LIN {X 0,Y 126.826,Z 270.322,A -85,B 0,C 180,E1 -25581.757,E2 -25581.757} C_VEL
LIN {X 0,Y 128.484,Z 273.393,A -85,B 0,C 180,E1 -25583.684,E2 -25583.684} C_VEL
LIN {X 0,Y 131.097,Z 275.877,A -85,B 0,C 180,E1 -25586.142,E2 -25586.142} C_VEL
LIN {X 0,Y 133.484,Z 279.395,A -85,B 0,C 180,E1 -25588.285,E2 -25588.285} C_VEL
LIN {X 0,Y 134.907,Z 280.969,A -85,B 0,C 180,E1 -25589.416,E2 -25589.416} C_VEL
LIN {X 0,Y 138.452,Z 286.009,A -85,B 0,C 180,E1 -25592.1,E2 -25592.1} C_VEL
LIN {X 0,Y 141.575,Z 290.551,A -85,B 0,C 180,E1 -25594.231,E2 -25594.231} C_VEL
LIN {X 0,Y 145.259,Z 296.604,A -85,B 0,C 180,E1 -25596.563,E2 -25596.563} C_VEL
LIN {X 0,Y 150.081,Z 307.019,A -85,B 0,C 180,E1 -25599.468,E2 -25599.468} C_VEL
LIN {X 0,Y 153.935,Z 317.286,A -85,B 0,C 180,E1 -25601.685,E2 -25601.685} C_VEL
LIN {X 0,Y 155.41,Z 322.258,A -85,B 0,C 180,E1 -25602.549,E2 -25602.549} C_VEL
LIN {X 0,Y 155.477,Z 325.681,A -85,B 0,C 180,E1 -25602.79,E2 -25602.79} C_VEL
LIN {X 0,Y 152.439,Z 367.811,A -85,B 0,C 180,E1 -25604.482,E2 -25604.482} C_VEL
LIN {X 0,Y 150.559,Z 380.968,A -85,B 0,C 180,E1 -25605.426,E2 -25605.426} C_VEL
LIN {X 0,Y 148.013,Z 393.091,A -85,B 0,C 180,E1 -25606.723,E2 -25606.723} C_VEL
LIN {X 0,Y 144.645,Z 405.228,A -85,B 0,C 180,E1 -25608.547,E2 -25608.547} C_VEL
LIN {X 0,Y 140.782,Z 416.789,A -85,B 0,C 180,E1 -25610.931,E2 -25610.931} C_VEL
LIN {X 0,Y 136.675,Z 427.192,A -85,B 0,C 180,E1 -25613.748,E2 -25613.748} C_VEL
LIN {X 0,Y 132.64,Z 436.533,A -85,B 0,C 180,E1 -25617.105,E2 -25617.105} C_VEL
LIN {X 0,Y 128.668,Z 445.603,A -85,B 0,C 180,E1 -25621.45,E2 -25621.45} C_VEL
LIN {X 0,Y 125.227,Z 452.89,A -85,B 0,C 180,E1 -25625.991,E2 -25625.991} C_VEL
LIN {X 0,Y 122.854,Z 457.8,A -85,B 0,C 180,E1 -25629.926,E2 -25629.926} C_VEL
LIN {X 0,Y 120.908,Z 462.575,A -85,B 0,C 180,E1 -25634.837,E2 -25634.837} C_VEL
LIN {X 0,Y 119.782,Z 466.223,A -85,B 0,C 180,E1 -25639.862,E2 -25639.862} C_VEL
LIN {X 0,Y 119.407,Z 468.103,A -85,B 0,C 180,E1 -25643.24,E2 -25643.24} C_VEL
LIN {X 0,Y 119.284,Z 469.509,A -85,B 0,C 180,E1 -25646.622,E2 -25646.622} C_VEL
LIN {X 0,Y 119.361,Z 470.506,A -85,B 0,C 180,E1 -25650,E2 -25650} C_VEL
LIN {X 0,Y 119.283,Z 471.098,A -85,B 0,C 180,E1 -25653.378,E2 -25653.378} C_VEL
LIN {X 0,Y 119.41,Z 471.3,A -85,B 0,C 180,E1 -25656.76,E2 -25656.76} C_VEL
LIN {X 0,Y 120.566,Z 470.457,A -85,B 0,C 180,E1 -25663.484,E2 -25663.484} C_VEL
LIN {X 0,Y 123.147,Z 468.068,A -85,B 0,C 180,E1 -25670.025,E2 -25670.025} C_VEL
LIN {X 0,Y 126.221,Z 465.155,A -85,B 0,C 180,E1 -25674.683,E2 -25674.683} C_VEL
LIN {X 0,Y 130.037,Z 461.227,A -85,B 0,C 180,E1 -25679.105,E2 -25679.105} C_VEL
LIN {X 0,Y 133.353,Z 457.578,A -85,B 0,C 180,E1 -25682.215,E2 -25682.215} C_VEL
LIN {X 0,Y 135.043,Z 454.869,A -85,B 0,C 180,E1 -25684.337,E2 -25684.337} C_VEL
LIN {X 0,Y 136.611,Z 450.087,A -85,B 0,C 180,E1 -25687.954,E2 -25687.954} C_VEL
LIN {X 0,Y 138.587,Z 444.753,A -85,B 0,C 180,E1 -25691.319,E2 -25691.319} C_VEL
LIN {X 0,Y 140.811,Z 441.114,A -85,B 0,C 180,E1 -25692.983,E2 -25692.983} C_VEL
LIN {X 0,Y 146.833,Z 432.313,A -85,B 0,C 180,E1 -25695.886,E2 -25695.886} C_VEL
LIN {X 0,Y 152.728,Z 422.206,A -85,B 0,C 180,E1 -25698.398,E2 -25698.398} C_VEL
LIN {X 0,Y 158.344,Z 410.772,A -85,B 0,C 180,E1 -25700.46,E2 -25700.46} C_VEL
LIN {X 0,Y 162.862,Z 399.545,A -85,B 0,C 180,E1 -25701.957,E2 -25701.957} C_VEL
LIN {X 0,Y 166.733,Z 386.906,A -85,B 0,C 180,E1 -25703.214,E2 -25703.214} C_VEL
LIN {X 0,Y 169.736,Z 373.483,A -85,B 0,C 180,E1 -25704.077,E2 -25704.077} C_VEL
LIN {X 0,Y 171.471,Z 360.998,A -85,B 0,C 180,E1 -25704.574,E2 -25704.574} C_VEL
LIN {X 0,Y 172.722,Z 344.57,A -85,B 0,C 180,E1 -25705.176,E2 -25705.176} C_VEL
LIN {X 0,Y 168.984,Z 334.445,A -85,B 0,C 180,E1 -25708.103,E2 -25708.103} C_VEL
LIN {X 0,Y 165.185,Z 325.649,A -85,B 0,C 180,E1 -25711.397,E2 -25711.397} C_VEL
LIN {X 0,Y 161.765,Z 318.418,A -85,B 0,C 180,E1 -25714.824,E2 -25714.824} C_VEL
LIN {X 0,Y 159.779,Z 315.16,A -85,B 0,C 180,E1 -25717.023,E2 -25717.023} C_VEL
LIN {X 0,Y 157.234,Z 311.251,A -85,B 0,C 180,E1 -25720.292,E2 -25720.292} C_VEL
LIN {X 0,Y 154.947,Z 307.802,A -85,B 0,C 180,E1 -25723.997,E2 -25723.997} C_VEL
LIN {X 0,Y 154.532,Z 306.974,A -85,B 0,C 180,E1 -25724.841,E2 -25724.841} C_VEL
LIN {X 0,Y 152.302,Z 304.116,A -85,B 0,C 180,E1 -25730.586,E2 -25730.586} C_VEL
LIN {X 0,Y 151.876,Z 301.949,A -85,B 0,C 180,E1 -25733.44,E2 -25733.44} C_VEL
LIN {X 0,Y 151.879,Z 301.933,A -85,B 0,C 180,E1 -25740.995,E2 -25740.995} C_VEL
LIN {X 0,Y 153.369,Z 305.636,A -85,B 0,C 180,E1 -25747.074,E2 -25747.074} C_VEL
LIN {X 0,Y 154.795,Z 307.238,A -85,B 0,C 180,E1 -25750.072,E2 -25750.072} C_VEL
LIN {X 0,Y 157.088,Z 310.973,A -85,B 0,C 180,E1 -25753.915,E2 -25753.915} C_VEL
LIN {X 0,Y 158.67,Z 313.546,A -85,B 0,C 180,E1 -25756.072,E2 -25756.072} C_VEL
LIN {X 0,Y 160.804,Z 316.708,A -85,B 0,C 180,E1 -25758.556,E2 -25758.556} C_VEL
LIN {X 0,Y 163.156,Z 320.534,A -85,B 0,C 180,E1 -25760.982,E2 -25760.982} C_VEL
LIN {X 0,Y 166.614,Z 326.408,A -85,B 0,C 180,E1 -25764.093,E2 -25764.093} C_VEL
LIN {X 0,Y 170.736,Z 334.213,A -85,B 0,C 180,E1 -25767.337,E2 -25767.337} C_VEL
LIN {X 0,Y 173.225,Z 339.607,A -85,B 0,C 180,E1 -25769.135,E2 -25769.135} C_VEL
LIN {X 0,Y 171.033,Z 362.908,A -85,B 0,C 180,E1 -25769.93,E2 -25769.93} C_VEL
LIN {X 0,Y 168.76,Z 375.767,A -85,B 0,C 180,E1 -25770.673,E2 -25770.673} C_VEL
LIN {X 0,Y 165.427,Z 388.725,A -85,B 0,C 180,E1 -25771.823,E2 -25771.823} C_VEL
LIN {X 0,Y 161.557,Z 399.746,A -85,B 0,C 180,E1 -25773.132,E2 -25773.132} C_VEL
LIN {X 0,Y 157.151,Z 409.955,A -85,B 0,C 180,E1 -25774.739,E2 -25774.739} C_VEL
LIN {X 0,Y 152.12,Z 419.837,A -85,B 0,C 180,E1 -25776.802,E2 -25776.802} C_VEL
LIN {X 0,Y 146.048,Z 430.047,A -85,B 0,C 180,E1 -25779.651,E2 -25779.651} C_VEL
LIN {X 0,Y 139.433,Z 439.163,A -85,B 0,C 180,E1 -25783.041,E2 -25783.041} C_VEL
LIN {X 0,Y 133.538,Z 446.491,A -85,B 0,C 180,E1 -25786.829,E2 -25786.829} C_VEL
LIN {X 0,Y 128.262,Z 452.341,A -85,B 0,C 180,E1 -25790.94,E2 -25790.94} C_VEL
LIN {X 0,Y 123.611,Z 456.926,A -85,B 0,C 180,E1 -25795.35,E2 -25795.35} C_VEL
LIN {X 0,Y 120.93,Z 459.336,A -85,B 0,C 180,E1 -25798.463,E2 -25798.463} C_VEL
LIN {X 0,Y 117.135,Z 462.465,A -85,B 0,C 180,E1 -25804.158,E2 -25804.158} C_VEL
LIN {X 0,Y 114.995,Z 463.953,A -85,B 0,C 180,E1 -25808.488,E2 -25808.488} C_VEL
LIN {X 0,Y 112.798,Z 464.935,A -85,B 0,C 180,E1 -25815.568,E2 -25815.568} C_VEL
LIN {X 0,Y 112.284,Z 464.849,A -85,B 0,C 180,E1 -25819.177,E2 -25819.177} C_VEL
LIN {X 0,Y 112.12,Z 464.344,A -85,B 0,C 180,E1 -25822.798,E2 -25822.798} C_VEL
LIN {X 0,Y 112.173,Z 463.43,A -85,B 0,C 180,E1 -25826.408,E2 -25826.408} C_VEL
LIN {X 0,Y 112.449,Z 462.131,A -85,B 0,C 180,E1 -25830,E2 -25830} C_VEL
LIN {X 0,Y 113.358,Z 459.394,A -85,B 0,C 180,E1 -25835.336,E2 -25835.336} C_VEL
LIN {X 0,Y 114.989,Z 455.651,A -85,B 0,C 180,E1 -25840.565,E2 -25840.565} C_VEL
LIN {X 0,Y 117.389,Z 450.796,A -85,B 0,C 180,E1 -25845.629,E2 -25845.629} C_VEL
LIN {X 0,Y 120.516,Z 444.687,A -85,B 0,C 180,E1 -25850.481,E2 -25850.481} C_VEL
LIN {X 0,Y 124.47,Z 437.084,A -85,B 0,C 180,E1 -25855.054,E2 -25855.054} C_VEL
LIN {X 0,Y 129.018,Z 427.533,A -85,B 0,C 180,E1 -25859.357,E2 -25859.357} C_VEL
LIN {X 0,Y 133.372,Z 417.674,A -85,B 0,C 180,E1 -25862.692,E2 -25862.692} C_VEL
LIN {X 0,Y 137.534,Z 406.586,A -85,B 0,C 180,E1 -25865.539,E2 -25865.539} C_VEL
LIN {X 0,Y 140.975,Z 395.728,A -85,B 0,C 180,E1 -25867.64,E2 -25867.64} C_VEL
LIN {X 0,Y 144.007,Z 383.744,A -85,B 0,C 180,E1 -25869.378,E2 -25869.378} C_VEL
LIN {X 0,Y 146.382,Z 371.309,A -85,B 0,C 180,E1 -25870.644,E2 -25870.644} C_VEL
LIN {X 0,Y 148,Z 357.95,A -85,B 0,C 180,E1 -25871.499,E2 -25871.499} C_VEL
LIN {X 0,Y 150.865,Z 319.683,A -85,B 0,C 180,E1 -25872.99,E2 -25872.99} C_VEL
LIN {X 0,Y 149.954,Z 317.15,A -85,B 0,C 180,E1 -25873.53,E2 -25873.53} C_VEL
LIN {X 0,Y 144.652,Z 306.547,A -85,B 0,C 180,E1 -25876.616,E2 -25876.616} C_VEL
LIN {X 0,Y 139.238,Z 297.373,A -85,B 0,C 180,E1 -25880.113,E2 -25880.113} C_VEL
LIN {X 0,Y 134.139,Z 289.816,A -85,B 0,C 180,E1 -25883.883,E2 -25883.883} C_VEL
LIN {X 0,Y 131.283,Z 285.807,A -85,B 0,C 180,E1 -25886.291,E2 -25886.291} C_VEL
LIN {X 0,Y 128.327,Z 281.654,A -85,B 0,C 180,E1 -25889.107,E2 -25889.107} C_VEL
LIN {X 0,Y 125.771,Z 278.792,A -85,B 0,C 180,E1 -25891.799,E2 -25891.799} C_VEL
LIN {X 0,Y 124.677,Z 276.71,A -85,B 0,C 180,E1 -25893.194,E2 -25893.194} C_VEL
LIN {X 0,Y 122.052,Z 274.673,A -85,B 0,C 180,E1 -25896.54,E2 -25896.54} C_VEL
LIN {X 0,Y 120.593,Z 271.942,A -85,B 0,C 180,E1 -25899.03,E2 -25899.03} C_VEL
LIN {X 0,Y 120.38,Z 271.211,A -85,B 0,C 180,E1 -25899.494,E2 -25899.494} C_VEL
LIN {X 0,Y 117.203,Z 269.28,A -85,B 0,C 180,E1 -25906.121,E2 -25906.121} C_VEL
LIN {X 0,Y 115.68,Z 266.37,A -85,B 0,C 180,E1 -25913.896,E2 -25913.896} C_VEL
LIN {X 0,Y 115.837,Z 265.042,A -85,B 0,C 180,E1 -25919.131,E2 -25919.131} C_VEL
LIN {X 0,Y 115.913,Z 265.227,A -85,B 0,C 180,E1 -25920.542,E2 -25920.542} C_VEL
LIN {X 0,Y 116.233,Z 267.39,A -85,B 0,C 180,E1 -25923.683,E2 -25923.683} C_VEL
LIN {X 0,Y 118.644,Z 270.26,A -85,B 0,C 180,E1 -25930.988,E2 -25930.988} C_VEL
LIN {X 0,Y 120.43,Z 271.31,A -85,B 0,C 180,E1 -25934.252,E2 -25934.252} C_VEL
LIN {X 0,Y 121.706,Z 274.109,A -85,B 0,C 180,E1 -25936.566,E2 -25936.566} C_VEL
LIN {X 0,Y 124.365,Z 276.547,A -85,B 0,C 180,E1 -25940.097,E2 -25940.097} C_VEL
LIN {X 0,Y 124.962,Z 277.268,A -85,B 0,C 180,E1 -25940.828,E2 -25940.828} C_VEL
LIN {X 0,Y 127.197,Z 280.647,A -85,B 0,C 180,E1 -25943.426,E2 -25943.426} C_VEL
LIN {X 0,Y 128.896,Z 282.384,A -85,B 0,C 180,E1 -25945.104,E2 -25945.104} C_VEL
LIN {X 0,Y 131.517,Z 286.037,A -85,B 0,C 180,E1 -25947.553,E2 -25947.553} C_VEL
LIN {X 0,Y 135.419,Z 291.569,A -85,B 0,C 180,E1 -25950.759,E2 -25950.759} C_VEL
LIN {X 0,Y 139.937,Z 298.477,A -85,B 0,C 180,E1 -25954.008,E2 -25954.008} C_VEL
LIN {X 0,Y 142.719,Z 303.955,A -85,B 0,C 180,E1 -25955.895,E2 -25955.895} C_VEL
LIN {X 0,Y 146.411,Z 312.55,A -85,B 0,C 180,E1 -25958.281,E2 -25958.281} C_VEL
LIN {X 0,Y 150.054,Z 323.022,A -85,B 0,C 180,E1 -25960.558,E2 -25960.558} C_VEL
LIN {X 0,Y 150.464,Z 324.735,A -85,B 0,C 180,E1 -25960.838,E2 -25960.838} C_VEL
LIN {X 0,Y 147.292,Z 367.734,A -85,B 0,C 180,E1 -25962.617,E2 -25962.617} C_VEL
LIN {X 0,Y 145.279,Z 381.195,A -85,B 0,C 180,E1 -25963.604,E2 -25963.604} C_VEL
LIN {X 0,Y 142.64,Z 393.137,A -85,B 0,C 180,E1 -25964.906,E2 -25964.906} C_VEL
LIN {X 0,Y 139.373,Z 404.404,A -85,B 0,C 180,E1 -25966.603,E2 -25966.603} C_VEL
LIN {X 0,Y 135.326,Z 416.082,A -85,B 0,C 180,E1 -25969.03,E2 -25969.03} C_VEL
LIN {X 0,Y 130.97,Z 426.57,A -85,B 0,C 180,E1 -25971.895,E2 -25971.895} C_VEL
LIN {X 0,Y 126.688,Z 436.011,A -85,B 0,C 180,E1 -25975.346,E2 -25975.346} C_VEL
LIN {X 0,Y 122.408,Z 445.135,A -85,B 0,C 180,E1 -25979.843,E2 -25979.843} C_VEL
LIN {X 0,Y 118.706,Z 452.469,A -85,B 0,C 180,E1 -25984.581,E2 -25984.581} C_VEL
LIN {X 0,Y 116.187,Z 457.424,A -85,B 0,C 180,E1 -25988.72,E2 -25988.72} C_VEL
LIN {X 0,Y 114.024,Z 462.236,A -85,B 0,C 180,E1 -25993.897,E2 -25993.897} C_VEL
LIN {X 0,Y 112.769,Z 465.921,A -85,B 0,C 180,E1 -25999.224,E2 -25999.224} C_VEL
LIN {X 0,Y 112.329,Z 467.821,A -85,B 0,C 180,E1 -26002.812,E2 -26002.812} C_VEL
LIN {X 0,Y 112.181,Z 469.257,A -85,B 0,C 180,E1 -26006.408,E2 -26006.408} C_VEL
LIN {X 0,Y 112.262,Z 470.27,A -85,B 0,C 180,E1 -26010,E2 -26010} C_VEL
LIN {X 0,Y 112.201,Z 470.878,A -85,B 0,C 180,E1 -26013.591,E2 -26013.591} C_VEL
LIN {X 0,Y 112.336,Z 471.098,A -85,B 0,C 180,E1 -26017.188,E2 -26017.188} C_VEL
LIN {X 0,Y 112.793,Z 470.9,A -85,B 0,C 180,E1 -26020.774,E2 -26020.774} C_VEL
LIN {X 0,Y 114.874,Z 469.316,A -85,B 0,C 180,E1 -26027.812,E2 -26027.812} C_VEL
LIN {X 0,Y 116.474,Z 467.943,A -85,B 0,C 180,E1 -26031.226,E2 -26031.226} C_VEL
LIN {X 0,Y 119.793,Z 465.063,A -85,B 0,C 180,E1 -26036.105,E2 -26036.105} C_VEL
LIN {X 0,Y 123.881,Z 461.17,A -85,B 0,C 180,E1 -26040.703,E2 -26040.703} C_VEL
LIN {X 0,Y 129.33,Z 455.389,A -85,B 0,C 180,E1 -26045.581,E2 -26045.581} C_VEL
LIN {X 0,Y 134.977,Z 448.685,A -85,B 0,C 180,E1 -26049.631,E2 -26049.631} C_VEL
LIN {X 0,Y 140.811,Z 441.114,A -85,B 0,C 180,E1 -26052.983,E2 -26052.983} C_VEL
LIN {X 0,Y 143.056,Z 437.279,A -85,B 0,C 180,E1 -26054.559,E2 -26054.559} C_VEL
LIN {X 0,Y 145.341,Z 430.766,A -85,B 0,C 180,E1 -26057.404,E2 -26057.404} C_VEL
LIN {X 0,Y 147.702,Z 423.796,A -85,B 0,C 180,E1 -26059.981,E2 -26059.981} C_VEL
LIN {X 0,Y 149.95,Z 419.15,A -85,B 0,C 180,E1 -26061.102,E2 -26061.102} C_VEL
LIN {X 0,Y 155.264,Z 408.282,A -85,B 0,C 180,E1 -26062.92,E2 -26062.92} C_VEL
LIN {X 0,Y 159.951,Z 396.309,A -85,B 0,C 180,E1 -26064.377,E2 -26064.377} C_VEL
LIN {X 0,Y 163.474,Z 384.532,A -85,B 0,C 180,E1 -26065.436,E2 -26065.436} C_VEL
LIN {X 0,Y 166.16,Z 372.192,A -85,B 0,C 180,E1 -26066.196,E2 -26066.196} C_VEL
LIN {X 0,Y 167.885,Z 359.393,A -85,B 0,C 180,E1 -26066.663,E2 -26066.663} C_VEL
LIN {X 0,Y 168.81,Z 347.255,A -85,B 0,C 180,E1 -26067.129,E2 -26067.129} C_VEL
LIN {X 0,Y 165.575,Z 338.228,A -85,B 0,C 180,E1 -26069.934,E2 -26069.934} C_VEL
LIN {X 0,Y 162.341,Z 330.413,A -85,B 0,C 180,E1 -26073.038,E2 -26073.038} C_VEL
LIN {X 0,Y 159.333,Z 323.765,A -85,B 0,C 180,E1 -26076.369,E2 -26076.369} C_VEL
LIN {X 0,Y 157.713,Z 321.142,A -85,B 0,C 180,E1 -26078.322,E2 -26078.322} C_VEL
LIN {X 0,Y 155.562,Z 317.639,A -85,B 0,C 180,E1 -26081.352,E2 -26081.352} C_VEL
LIN {X 0,Y 153.494,Z 314.14,A -85,B 0,C 180,E1 -26085.075,E2 -26085.075} C_VEL
LIN {X 0,Y 151.207,Z 310.7,A -85,B 0,C 180,E1 -26091.566,E2 -26091.566} C_VEL
LIN {X 0,Y 150.946,Z 308.985,A -85,B 0,C 180,E1 -26093.819,E2 -26093.819} C_VEL
LIN {X 0,Y 150.922,Z 308.838,A -85,B 0,C 180,E1 -26100.334,E2 -26100.334} C_VEL
LIN {X 0,Y 152.671,Z 313.002,A -85,B 0,C 180,E1 -26107.538,E2 -26107.538} C_VEL
LIN {X 0,Y 153.606,Z 314.216,A -85,B 0,C 180,E1 -26109.56,E2 -26109.56} C_VEL
LIN {X 0,Y 156.387,Z 318.86,A -85,B 0,C 180,E1 -26114.29,E2 -26114.29} C_VEL
LIN {X 0,Y 159.037,Z 323.21,A -85,B 0,C 180,E1 -26117.708,E2 -26117.708} C_VEL
LIN {X 0,Y 161.398,Z 327.222,A -85,B 0,C 180,E1 -26120.283,E2 -26120.283} C_VEL
LIN {X 0,Y 165.141,Z 334.046,A -85,B 0,C 180,E1 -26123.806,E2 -26123.806} C_VEL
LIN {X 0,Y 169.184,Z 342.339,A -85,B 0,C 180,E1 -26127.107,E2 -26127.107} C_VEL
LIN {X 0,Y 169.176,Z 344.32,A -85,B 0,C 180,E1 -26127.267,E2 -26127.267} C_VEL
LIN {X 0,Y 167.199,Z 363.569,A -85,B 0,C 180,E1 -26127.913,E2 -26127.913} C_VEL
LIN {X 0,Y 164.786,Z 376.603,A -85,B 0,C 180,E1 -26128.672,E2 -26128.672} C_VEL
LIN {X 0,Y 161.437,Z 389.043,A -85,B 0,C 180,E1 -26129.777,E2 -26129.777} C_VEL
LIN {X 0,Y 157.1,Z 400.836,A -85,B 0,C 180,E1 -26131.177,E2 -26131.177} C_VEL
LIN {X 0,Y 151.884,Z 412.18,A -85,B 0,C 180,E1 -26132.998,E2 -26132.998} C_VEL
LIN {X 0,Y 146.295,Z 422.366,A -85,B 0,C 180,E1 -26135.246,E2 -26135.246} C_VEL
LIN {X 0,Y 140.393,Z 431.524,A -85,B 0,C 180,E1 -26137.96,E2 -26137.96} C_VEL
LIN {X 0,Y 133.53,Z 440.421,A -85,B 0,C 180,E1 -26141.409,E2 -26141.409} C_VEL
LIN {X 0,Y 127.402,Z 447.526,A -85,B 0,C 180,E1 -26145.291,E2 -26145.291} C_VEL
LIN {X 0,Y 121.019,Z 453.995,A -85,B 0,C 180,E1 -26150.297,E2 -26150.297} C_VEL
LIN {X 0,Y 116.259,Z 458.238,A -85,B 0,C 180,E1 -26154.95,E2 -26154.95} C_VEL
LIN {X 0,Y 112.336,Z 461.4,A -85,B 0,C 180,E1 -26159.967,E2 -26159.967} C_VEL
LIN {X 0,Y 110.165,Z 462.965,A -85,B 0,C 180,E1 -26163.476,E2 -26163.476} C_VEL
LIN {X 0,Y 108.336,Z 464.107,A -85,B 0,C 180,E1 -26167.093,E2 -26167.093} C_VEL
LIN {X 0,Y 105.858,Z 465.125,A -85,B 0,C 180,E1 -26174.6,E2 -26174.6} C_VEL
LIN {X 0,Y 105.259,Z 465.056,A -85,B 0,C 180,E1 -26178.445,E2 -26178.445} C_VEL
LIN {X 0,Y 105.03,Z 464.586,A -85,B 0,C 180,E1 -26182.309,E2 -26182.309} C_VEL
LIN {X 0,Y 105.079,Z 463.689,A -85,B 0,C 180,E1 -26186.165,E2 -26186.165} C_VEL
LIN {X 0,Y 105.43,Z 462.132,A -85,B 0,C 180,E1 -26190.725,E2 -26190.725} C_VEL
LIN {X 0,Y 106.795,Z 458.606,A -85,B 0,C 180,E1 -26197.563,E2 -26197.563} C_VEL
LIN {X 0,Y 108.806,Z 454.547,A -85,B 0,C 180,E1 -26203.066,E2 -26203.066} C_VEL
LIN {X 0,Y 112.136,Z 448.329,A -85,B 0,C 180,E1 -26209.21,E2 -26209.21} C_VEL
LIN {X 0,Y 115.938,Z 441.559,A -85,B 0,C 180,E1 -26214.153,E2 -26214.153} C_VEL
LIN {X 0,Y 120.446,Z 433.123,A -85,B 0,C 180,E1 -26218.777,E2 -26218.777} C_VEL
LIN {X 0,Y 124.709,Z 424.451,A -85,B 0,C 180,E1 -26222.369,E2 -26222.369} C_VEL
LIN {X 0,Y 129.384,Z 413.777,A -85,B 0,C 180,E1 -26225.727,E2 -26225.727} C_VEL
LIN {X 0,Y 133.397,Z 403.133,A -85,B 0,C 180,E1 -26228.247,E2 -26228.247} C_VEL
LIN {X 0,Y 137.046,Z 391.213,A -85,B 0,C 180,E1 -26230.349,E2 -26230.349} C_VEL
LIN {X 0,Y 140.134,Z 378.16,A -85,B 0,C 180,E1 -26232.006,E2 -26232.006} C_VEL
LIN {X 0,Y 142.275,Z 365.227,A -85,B 0,C 180,E1 -26233.092,E2 -26233.092} C_VEL
LIN {X 0,Y 143.874,Z 347.807,A -85,B 0,C 180,E1 -26233.919,E2 -26233.919} C_VEL
LIN {X 0,Y 145.874,Z 321.687,A -85,B 0,C 180,E1 -26234.938,E2 -26234.938} C_VEL
LIN {X 0,Y 140.887,Z 311.337,A -85,B 0,C 180,E1 -26238.086,E2 -26238.086} C_VEL
LIN {X 0,Y 135.772,Z 302.426,A -85,B 0,C 180,E1 -26241.673,E2 -26241.673} C_VEL
LIN {X 0,Y 131.221,Z 295.406,A -85,B 0,C 180,E1 -26245.333,E2 -26245.333} C_VEL
LIN {X 0,Y 128.587,Z 291.604,A -85,B 0,C 180,E1 -26247.74,E2 -26247.74} C_VEL
LIN {X 0,Y 125.858,Z 287.692,A -85,B 0,C 180,E1 -26250.561,E2 -26250.561} C_VEL
LIN {X 0,Y 123.364,Z 284.409,A -85,B 0,C 180,E1 -26253.495,E2 -26253.495} C_VEL
LIN {X 0,Y 122.592,Z 283.199,A -85,B 0,C 180,E1 -26254.534,E2 -26254.534} C_VEL
LIN {X 0,Y 120.063,Z 280.701,A -85,B 0,C 180,E1 -26258.155,E2 -26258.155} C_VEL
LIN {X 0,Y 118.829,Z 278.036,A -85,B 0,C 180,E1 -26260.568,E2 -26260.568} C_VEL
LIN {X 0,Y 116.031,Z 276.032,A -85,B 0,C 180,E1 -26267.016,E2 -26267.016} C_VEL
LIN {X 0,Y 114.742,Z 272.986,A -85,B 0,C 180,E1 -26275.609,E2 -26275.609} C_VEL
LIN {X 0,Y 114.838,Z 272.283,A -85,B 0,C 180,E1 -26278.246,E2 -26278.246} C_VEL
LIN {X 0,Y 114.961,Z 272.627,A -85,B 0,C 180,E1 -26280.219,E2 -26280.219} C_VEL
LIN {X 0,Y 115.566,Z 275.123,A -85,B 0,C 180,E1 -26284.796,E2 -26284.796} C_VEL
LIN {X 0,Y 118.902,Z 278.148,A -85,B 0,C 180,E1 -26293.226,E2 -26293.226} C_VEL
LIN {X 0,Y 120.308,Z 280.999,A -85,B 0,C 180,E1 -26295.892,E2 -26295.892} C_VEL
LIN {X 0,Y 122.977,Z 283.651,A -85,B 0,C 180,E1 -26299.618,E2 -26299.618} C_VEL
LIN {X 0,Y 125.304,Z 287.177,A -85,B 0,C 180,E1 -26302.498,E2 -26302.498} C_VEL
LIN {X 0,Y 126.661,Z 288.694,A -85,B 0,C 180,E1 -26303.938,E2 -26303.938} C_VEL
LIN {X 0,Y 130.147,Z 293.716,A -85,B 0,C 180,E1 -26307.35,E2 -26307.35} C_VEL
LIN {X 0,Y 134.409,Z 300.046,A -85,B 0,C 180,E1 -26310.914,E2 -26310.914} C_VEL
LIN {X 0,Y 138.019,Z 306.426,A -85,B 0,C 180,E1 -26313.625,E2 -26313.625} C_VEL
LIN {X 0,Y 142.031,Z 315.996,A -85,B 0,C 180,E1 -26316.498,E2 -26316.498} C_VEL
LIN {X 0,Y 145.294,Z 325.657,A -85,B 0,C 180,E1 -26318.741,E2 -26318.741} C_VEL
LIN {X 0,Y 145.554,Z 327.024,A -85,B 0,C 180,E1 -26318.954,E2 -26318.954} C_VEL
LIN {X 0,Y 142.298,Z 367.725,A -85,B 0,C 180,E1 -26320.624,E2 -26320.624} C_VEL
LIN {X 0,Y 140.165,Z 381.308,A -85,B 0,C 180,E1 -26321.633,E2 -26321.633} C_VEL
LIN {X 0,Y 137.425,Z 393.168,A -85,B 0,C 180,E1 -26322.95,E2 -26322.95} C_VEL
LIN {X 0,Y 133.749,Z 405.168,A -85,B 0,C 180,E1 -26324.816,E2 -26324.816} C_VEL
LIN {X 0,Y 129.498,Z 416.667,A -85,B 0,C 180,E1 -26327.282,E2 -26327.282} C_VEL
LIN {X 0,Y 124.945,Z 427.017,A -85,B 0,C 180,E1 -26330.221,E2 -26330.221} C_VEL
LIN {X 0,Y 120.043,Z 437.132,A -85,B 0,C 180,E1 -26334.165,E2 -26334.165} C_VEL
LIN {X 0,Y 116.234,Z 444.69,A -85,B 0,C 180,E1 -26338.077,E2 -26338.077} C_VEL
LIN {X 0,Y 112.88,Z 450.921,A -85,B 0,C 180,E1 -26342.163,E2 -26342.163} C_VEL
LIN {X 0,Y 109.581,Z 457.048,A -85,B 0,C 180,E1 -26347.368,E2 -26347.368} C_VEL
LIN {X 0,Y 107.182,Z 461.898,A -85,B 0,C 180,E1 -26352.839,E2 -26352.839} C_VEL
LIN {X 0,Y 105.788,Z 465.619,A -85,B 0,C 180,E1 -26358.504,E2 -26358.504} C_VEL
LIN {X 0,Y 105.272,Z 467.536,A -85,B 0,C 180,E1 -26362.327,E2 -26362.327} C_VEL
LIN {X 0,Y 105.097,Z 469.005,A -85,B 0,C 180,E1 -26366.166,E2 -26366.166} C_VEL
LIN {X 0,Y 105.175,Z 470.034,A -85,B 0,C 180,E1 -26370,E2 -26370} C_VEL
LIN {X 0,Y 105.11,Z 470.657,A -85,B 0,C 180,E1 -26373.834,E2 -26373.834} C_VEL
LIN {X 0,Y 105.279,Z 470.893,A -85,B 0,C 180,E1 -26377.673,E2 -26377.673} C_VEL
LIN {X 0,Y 105.813,Z 470.727,A -85,B 0,C 180,E1 -26381.494,E2 -26381.494} C_VEL
LIN {X 0,Y 108.094,Z 469.174,A -85,B 0,C 180,E1 -26388.971,E2 -26388.971} C_VEL
LIN {X 0,Y 109.864,Z 467.818,A -85,B 0,C 180,E1 -26392.571,E2 -26392.571} C_VEL
LIN {X 0,Y 113.445,Z 464.972,A -85,B 0,C 180,E1 -26397.686,E2 -26397.686} C_VEL
LIN {X 0,Y 117.83,Z 461.116,A -85,B 0,C 180,E1 -26402.467,E2 -26402.467} C_VEL
LIN {X 0,Y 123.398,Z 455.619,A -85,B 0,C 180,E1 -26407.324,E2 -26407.324} C_VEL
LIN {X 0,Y 129.579,Z 448.734,A -85,B 0,C 180,E1 -26411.637,E2 -26411.637} C_VEL
LIN {X 0,Y 136.123,Z 440.679,A -85,B 0,C 180,E1 -26415.228,E2 -26415.228} C_VEL
LIN {X 0,Y 141.992,Z 432.472,A -85,B 0,C 180,E1 -26417.939,E2 -26417.939} C_VEL
LIN {X 0,Y 148.123,Z 422.467,A -85,B 0,C 180,E1 -26420.445,E2 -26420.445} C_VEL
LIN {X 0,Y 149.95,Z 419.15,A -85,B 0,C 180,E1 -26421.102,E2 -26421.102} C_VEL
LIN {X 0,Y 151.272,Z 415.992,A -85,B 0,C 180,E1 -26421.879,E2 -26421.879} C_VEL
LIN {X 0,Y 152.049,Z 411.02,A -85,B 0,C 180,E1 -26423.59,E2 -26423.59} C_VEL
LIN {X 0,Y 152.725,Z 405.872,A -85,B 0,C 180,E1 -26425.227,E2 -26425.227} C_VEL
LIN {X 0,Y 153.819,Z 402.439,A -85,B 0,C 180,E1 -26425.866,E2 -26425.866} C_VEL
LIN {X 0,Y 158.343,Z 389.577,A -85,B 0,C 180,E1 -26427.197,E2 -26427.197} C_VEL
LIN {X 0,Y 161.594,Z 377.163,A -85,B 0,C 180,E1 -26428.077,E2 -26428.077} C_VEL
LIN {X 0,Y 163.819,Z 364.366,A -85,B 0,C 180,E1 -26428.632,E2 -26428.632} C_VEL
LIN {X 0,Y 165.152,Z 350.219,A -85,B 0,C 180,E1 -26429.116,E2 -26429.116} C_VEL
LIN {X 0,Y 162.501,Z 342.549,A -85,B 0,C 180,E1 -26431.67,E2 -26431.67} C_VEL
LIN {X 0,Y 159.515,Z 334.863,A -85,B 0,C 180,E1 -26434.876,E2 -26434.876} C_VEL
LIN {X 0,Y 157.119,Z 329.345,A -85,B 0,C 180,E1 -26437.827,E2 -26437.827} C_VEL
LIN {X 0,Y 154.158,Z 324.328,A -85,B 0,C 180,E1 -26442.086,E2 -26442.086} C_VEL
LIN {X 0,Y 152.056,Z 320.673,A -85,B 0,C 180,E1 -26446.203,E2 -26446.203} C_VEL
LIN {X 0,Y 150.198,Z 317.48,A -85,B 0,C 180,E1 -26452.269,E2 -26452.269} C_VEL
LIN {X 0,Y 150.017,Z 316.064,A -85,B 0,C 180,E1 -26454.203,E2 -26454.203} C_VEL
LIN {X 0,Y 150.037,Z 316.031,A -85,B 0,C 180,E1 -26460.336,E2 -26460.336} C_VEL
LIN {X 0,Y 151.622,Z 319.95,A -85,B 0,C 180,E1 -26467.156,E2 -26467.156} C_VEL
LIN {X 0,Y 152.358,Z 320.985,A -85,B 0,C 180,E1 -26468.862,E2 -26468.862} C_VEL
LIN {X 0,Y 154.81,Z 325.331,A -85,B 0,C 180,E1 -26473.371,E2 -26473.371} C_VEL
LIN {X 0,Y 157.484,Z 329.95,A -85,B 0,C 180,E1 -26477.051,E2 -26477.051} C_VEL
LIN {X 0,Y 160.28,Z 335.032,A -85,B 0,C 180,E1 -26480.222,E2 -26480.222} C_VEL
LIN {X 0,Y 163.88,Z 342.223,A -85,B 0,C 180,E1 -26483.712,E2 -26483.712} C_VEL
LIN {X 0,Y 165.532,Z 345.865,A -85,B 0,C 180,E1 -26485.163,E2 -26485.163} C_VEL
LIN {X 0,Y 163.511,Z 364.721,A -85,B 0,C 180,E1 -26485.827,E2 -26485.827} C_VEL
LIN {X 0,Y 160.945,Z 377.768,A -85,B 0,C 180,E1 -26486.598,E2 -26486.598} C_VEL
LIN {X 0,Y 157.302,Z 390.362,A -85,B 0,C 180,E1 -26487.725,E2 -26487.725} C_VEL
LIN {X 0,Y 152.846,Z 401.928,A -85,B 0,C 180,E1 -26489.116,E2 -26489.116} C_VEL
LIN {X 0,Y 147.445,Z 413.097,A -85,B 0,C 180,E1 -26490.91,E2 -26490.91} C_VEL
LIN {X 0,Y 142.139,Z 422.353,A -85,B 0,C 180,E1 -26492.949,E2 -26492.949} C_VEL
LIN {X 0,Y 136.108,Z 431.361,A -85,B 0,C 180,E1 -26495.584,E2 -26495.584} C_VEL
LIN {X 0,Y 130.065,Z 438.958,A -85,B 0,C 180,E1 -26498.418,E2 -26498.418} C_VEL
LIN {X 0,Y 123.431,Z 446.392,A -85,B 0,C 180,E1 -26502.251,E2 -26502.251} C_VEL
LIN {X 0,Y 117.41,Z 452.337,A -85,B 0,C 180,E1 -26506.499,E2 -26506.499} C_VEL
LIN {X 0,Y 112.051,Z 457.011,A -85,B 0,C 180,E1 -26511.155,E2 -26511.155} C_VEL
LIN {X 0,Y 107.479,Z 460.56,A -85,B 0,C 180,E1 -26516.233,E2 -26516.233} C_VEL
LIN {X 0,Y 103.786,Z 463.083,A -85,B 0,C 180,E1 -26521.705,E2 -26521.705} C_VEL
LIN {X 0,Y 101.752,Z 464.255,A -85,B 0,C 180,E1 -26525.517,E2 -26525.517} C_VEL
LIN {X 0,Y 98.952,Z 465.315,A -85,B 0,C 180,E1 -26533.495,E2 -26533.495} C_VEL
LIN {X 0,Y 98.264,Z 465.263,A -85,B 0,C 180,E1 -26537.61,E2 -26537.61} C_VEL
LIN {X 0,Y 97.94,Z 464.822,A -85,B 0,C 180,E1 -26541.748,E2 -26541.748} C_VEL
LIN {X 0,Y 97.958,Z 463.949,A -85,B 0,C 180,E1 -26545.886,E2 -26545.886} C_VEL
LIN {X 0,Y 98.431,Z 462.114,A -85,B 0,C 180,E1 -26551.584,E2 -26551.584} C_VEL
LIN {X 0,Y 99.77,Z 458.938,A -85,B 0,C 180,E1 -26558.099,E2 -26558.099} C_VEL
LIN {X 0,Y 101.929,Z 454.919,A -85,B 0,C 180,E1 -26563.965,E2 -26563.965} C_VEL
LIN {X 0,Y 105.486,Z 448.746,A -85,B 0,C 180,E1 -26570.474,E2 -26570.474} C_VEL
LIN {X 0,Y 109.509,Z 442.025,A -85,B 0,C 180,E1 -26575.67,E2 -26575.67} C_VEL
LIN {X 0,Y 114.311,Z 433.673,A -85,B 0,C 180,E1 -26580.48,E2 -26580.48} C_VEL
LIN {X 0,Y 118.807,Z 425.073,A -85,B 0,C 180,E1 -26584.192,E2 -26584.192} C_VEL
LIN {X 0,Y 123.713,Z 414.487,A -85,B 0,C 180,E1 -26587.64,E2 -26587.64} C_VEL
LIN {X 0,Y 127.915,Z 403.968,A -85,B 0,C 180,E1 -26590.209,E2 -26590.209} C_VEL
LIN {X 0,Y 131.748,Z 392.277,A -85,B 0,C 180,E1 -26592.335,E2 -26592.335} C_VEL
LIN {X 0,Y 134.991,Z 379.433,A -85,B 0,C 180,E1 -26594.015,E2 -26594.015} C_VEL
LIN {X 0,Y 137.364,Z 366.121,A -85,B 0,C 180,E1 -26595.189,E2 -26595.189} C_VEL
LIN {X 0,Y 138.972,Z 350.08,A -85,B 0,C 180,E1 -26595.975,E2 -26595.975} C_VEL
LIN {X 0,Y 141.052,Z 324.264,A -85,B 0,C 180,E1 -26596.98,E2 -26596.98} C_VEL
LIN {X 0,Y 136.315,Z 314.404,A -85,B 0,C 180,E1 -26600.293,E2 -26600.293} C_VEL
LIN {X 0,Y 131.443,Z 305.718,A -85,B 0,C 180,E1 -26604.133,E2 -26604.133} C_VEL
LIN {X 0,Y 126.82,Z 298.42,A -85,B 0,C 180,E1 -26608.407,E2 -26608.407} C_VEL
LIN {X 0,Y 123.714,Z 293.998,A -85,B 0,C 180,E1 -26611.794,E2 -26611.794} C_VEL
LIN {X 0,Y 120.737,Z 289.719,A -85,B 0,C 180,E1 -26615.71,E2 -26615.71} C_VEL
LIN {X 0,Y 118.312,Z 286.978,A -85,B 0,C 180,E1 -26619.551,E2 -26619.551} C_VEL
LIN {X 0,Y 117.292,Z 284.835,A -85,B 0,C 180,E1 -26621.727,E2 -26621.727} C_VEL
LIN {X 0,Y 114.912,Z 282.866,A -85,B 0,C 180,E1 -26627.819,E2 -26627.819} C_VEL
LIN {X 0,Y 113.871,Z 279.882,A -85,B 0,C 180,E1 -26636.461,E2 -26636.461} C_VEL
LIN {X 0,Y 114.049,Z 280.09,A -85,B 0,C 180,E1 -26640.275,E2 -26640.275} C_VEL
LIN {X 0,Y 115.275,Z 283.135,A -85,B 0,C 180,E1 -26647.003,E2 -26647.003} C_VEL
LIN {X 0,Y 117.467,Z 284.985,A -85,B 0,C 180,E1 -26652.269,E2 -26652.269} C_VEL
LIN {X 0,Y 119.143,Z 288.136,A -85,B 0,C 180,E1 -26655.558,E2 -26655.558} C_VEL
LIN {X 0,Y 121.22,Z 290.346,A -85,B 0,C 180,E1 -26658.622,E2 -26658.622} C_VEL
LIN {X 0,Y 123.747,Z 294.017,A -85,B 0,C 180,E1 -26661.888,E2 -26661.888} C_VEL
LIN {X 0,Y 124.991,Z 295.832,A -85,B 0,C 180,E1 -26663.315,E2 -26663.315} C_VEL
LIN {X 0,Y 127.818,Z 299.964,A -85,B 0,C 180,E1 -26666.233,E2 -26666.233} C_VEL
LIN {X 0,Y 131.725,Z 306.128,A -85,B 0,C 180,E1 -26669.745,E2 -26669.745} C_VEL
LIN {X 0,Y 134.87,Z 312.023,A -85,B 0,C 180,E1 -26672.298,E2 -26672.298} C_VEL
LIN {X 0,Y 138.38,Z 321.061,A -85,B 0,C 180,E1 -26675.05,E2 -26675.05} C_VEL
LIN {X 0,Y 140.714,Z 328.397,A -85,B 0,C 180,E1 -26676.823,E2 -26676.823} C_VEL
LIN {X 0,Y 137.577,Z 367.067,A -85,B 0,C 180,E1 -26678.451,E2 -26678.451} C_VEL
LIN {X 0,Y 135.363,Z 380.646,A -85,B 0,C 180,E1 -26679.439,E2 -26679.439} C_VEL
LIN {X 0,Y 132.375,Z 393.188,A -85,B 0,C 180,E1 -26680.839,E2 -26680.839} C_VEL
LIN {X 0,Y 128.812,Z 404.334,A -85,B 0,C 180,E1 -26682.561,E2 -26682.561} C_VEL
LIN {X 0,Y 124.345,Z 415.95,A -85,B 0,C 180,E1 -26685.049,E2 -26685.049} C_VEL
LIN {X 0,Y 119.567,Z 426.396,A -85,B 0,C 180,E1 -26688.04,E2 -26688.04} C_VEL
LIN {X 0,Y 115.227,Z 434.938,A -85,B 0,C 180,E1 -26691.305,E2 -26691.305} C_VEL
LIN {X 0,Y 110.36,Z 443.871,A -85,B 0,C 180,E1 -26695.88,E2 -26695.88} C_VEL
LIN {X 0,Y 107.374,Z 449.359,A -85,B 0,C 180,E1 -26699.518,E2 -26699.518} C_VEL
LIN {X 0,Y 104.16,Z 454.775,A -85,B 0,C 180,E1 -26703.987,E2 -26703.987} C_VEL
LIN {X 0,Y 101.096,Z 460.074,A -85,B 0,C 180,E1 -26709.66,E2 -26709.66} C_VEL
LIN {X 0,Y 99.213,Z 464.198,A -85,B 0,C 180,E1 -26715.645,E2 -26715.645} C_VEL
LIN {X 0,Y 98.218,Z 467.25,A -85,B 0,C 180,E1 -26721.772,E2 -26721.772} C_VEL
LIN {X 0,Y 98.012,Z 468.752,A -85,B 0,C 180,E1 -26725.888,E2 -26725.888} C_VEL
LIN {X 0,Y 98.079,Z 469.798,A -85,B 0,C 180,E1 -26730,E2 -26730} C_VEL
LIN {X 0,Y 98.021,Z 470.437,A -85,B 0,C 180,E1 -26734.112,E2 -26734.112} C_VEL
LIN {X 0,Y 98.247,Z 470.689,A -85,B 0,C 180,E1 -26738.226,E2 -26738.226} C_VEL
LIN {X 0,Y 98.834,Z 470.549,A -85,B 0,C 180,E1 -26742.318,E2 -26742.318} C_VEL
LIN {X 0,Y 101.367,Z 469.033,A -85,B 0,C 180,E1 -26750.283,E2 -26750.283} C_VEL
LIN {X 0,Y 103.329,Z 467.694,A -85,B 0,C 180,E1 -26754.085,E2 -26754.085} C_VEL
LIN {X 0,Y 107.195,Z 464.882,A -85,B 0,C 180,E1 -26759.454,E2 -26759.454} C_VEL
LIN {X 0,Y 111.902,Z 461.061,A -85,B 0,C 180,E1 -26764.42,E2 -26764.42} C_VEL
LIN {X 0,Y 117.249,Z 456.134,A -85,B 0,C 180,E1 -26769.002,E2 -26769.002} C_VEL
LIN {X 0,Y 123.279,Z 449.949,A -85,B 0,C 180,E1 -26773.165,E2 -26773.165} C_VEL
LIN {X 0,Y 130.019,Z 442.264,A -85,B 0,C 180,E1 -26776.863,E2 -26776.863} C_VEL
LIN {X 0,Y 137.336,Z 432.632,A -85,B 0,C 180,E1 -26780.14,E2 -26780.14} C_VEL
LIN {X 0,Y 143.72,Z 422.707,A -85,B 0,C 180,E1 -26782.621,E2 -26782.621} C_VEL
LIN {X 0,Y 149.738,Z 411.515,A -85,B 0,C 180,E1 -26784.637,E2 -26784.637} C_VEL
LIN {X 0,Y 153.819,Z 402.439,A -85,B 0,C 180,E1 -26785.866,E2 -26785.866} C_VEL
LIN {X 0,Y 155.562,Z 397.209,A -85,B 0,C 180,E1 -26786.649,E2 -26786.649} C_VEL
LIN {X 0,Y 157.023,Z 388.583,A -85,B 0,C 180,E1 -26788.36,E2 -26788.36} C_VEL
LIN {X 0,Y 157.992,Z 379.693,A -85,B 0,C 180,E1 -26789.921,E2 -26789.921} C_VEL
LIN {X 0,Y 158.888,Z 374.047,A -85,B 0,C 180,E1 -26790.459,E2 -26790.459} C_VEL
LIN {X 0,Y 160.954,Z 360.844,A -85,B 0,C 180,E1 -26790.962,E2 -26790.962} C_VEL
LIN {X 0,Y 161.642,Z 353.043,A -85,B 0,C 180,E1 -26791.251,E2 -26791.251} C_VEL
LIN {X 0,Y 159.037,Z 345.172,A -85,B 0,C 180,E1 -26794.11,E2 -26794.11} C_VEL
LIN {X 0,Y 156.174,Z 337.638,A -85,B 0,C 180,E1 -26797.685,E2 -26797.685} C_VEL
LIN {X 0,Y 154.94,Z 334.831,A -85,B 0,C 180,E1 -26799.421,E2 -26799.421} C_VEL
LIN {X 0,Y 152.714,Z 330.951,A -85,B 0,C 180,E1 -26802.94,E2 -26802.94} C_VEL
LIN {X 0,Y 150.875,Z 327.496,A -85,B 0,C 180,E1 -26806.857,E2 -26806.857} C_VEL
LIN {X 0,Y 149.223,Z 324.292,A -85,B 0,C 180,E1 -26812.899,E2 -26812.899} C_VEL
LIN {X 0,Y 149.101,Z 323.097,A -85,B 0,C 180,E1 -26814.591,E2 -26814.591} C_VEL
LIN {X 0,Y 149.122,Z 323.087,A -85,B 0,C 180,E1 -26820,E2 -26820} C_VEL
LIN {X 0,Y 150.587,Z 326.893,A -85,B 0,C 180,E1 -26826.785,E2 -26826.785} C_VEL
LIN {X 0,Y 151.222,Z 327.958,A -85,B 0,C 180,E1 -26828.372,E2 -26828.372} C_VEL
LIN {X 0,Y 153.377,Z 332.037,A -85,B 0,C 180,E1 -26832.614,E2 -26832.614} C_VEL
LIN {X 0,Y 155.523,Z 335.934,A -85,B 0,C 180,E1 -26835.816,E2 -26835.816} C_VEL
LIN {X 0,Y 158.205,Z 341.102,A -85,B 0,C 180,E1 -26839.125,E2 -26839.125} C_VEL
LIN {X 0,Y 161.827,Z 348.848,A -85,B 0,C 180,E1 -26842.892,E2 -26842.892} C_VEL
LIN {X 0,Y 162.014,Z 349.294,A -85,B 0,C 180,E1 -26843.073,E2 -26843.073} C_VEL
LIN {X 0,Y 160.067,Z 365.737,A -85,B 0,C 180,E1 -26843.636,E2 -26843.636} C_VEL
LIN {X 0,Y 157.618,Z 377.692,A -85,B 0,C 180,E1 -26844.336,E2 -26844.336} C_VEL
LIN {X 0,Y 154.113,Z 389.69,A -85,B 0,C 180,E1 -26845.377,E2 -26845.377} C_VEL
LIN {X 0,Y 149.489,Z 401.43,A -85,B 0,C 180,E1 -26846.714,E2 -26846.714} C_VEL
LIN {X 0,Y 143.895,Z 412.735,A -85,B 0,C 180,E1 -26848.461,E2 -26848.461} C_VEL
LIN {X 0,Y 137.782,Z 422.98,A -85,B 0,C 180,E1 -26850.67,E2 -26850.67} C_VEL
LIN {X 0,Y 130.775,Z 432.835,A -85,B 0,C 180,E1 -26853.593,E2 -26853.593} C_VEL
LIN {X 0,Y 124.506,Z 440.216,A -85,B 0,C 180,E1 -26856.451,E2 -26856.451} C_VEL
LIN {X 0,Y 117.588,Z 447.462,A -85,B 0,C 180,E1 -26860.355,E2 -26860.355} C_VEL
LIN {X 0,Y 112.246,Z 452.38,A -85,B 0,C 180,E1 -26864.007,E2 -26864.007} C_VEL
LIN {X 0,Y 106.539,Z 457.051,A -85,B 0,C 180,E1 -26868.726,E2 -26868.726} C_VEL
LIN {X 0,Y 101.576,Z 460.64,A -85,B 0,C 180,E1 -26873.977,E2 -26873.977} C_VEL
LIN {X 0,Y 97.248,Z 463.36,A -85,B 0,C 180,E1 -26880.14,E2 -26880.14} C_VEL
LIN {X 0,Y 93.452,Z 465.153,A -85,B 0,C 180,E1 -26887.912,E2 -26887.912} C_VEL
LIN {X 0,Y 91.261,Z 465.47,A -85,B 0,C 180,E1 -26896.642,E2 -26896.642} C_VEL
LIN {X 0,Y 90.879,Z 465.052,A -85,B 0,C 180,E1 -26901.102,E2 -26901.102} C_VEL
LIN {X 0,Y 90.864,Z 464.207,A -85,B 0,C 180,E1 -26905.564,E2 -26905.564} C_VEL
LIN {X 0,Y 91.467,Z 462.011,A -85,B 0,C 180,E1 -26912.7,E2 -26912.7} C_VEL
LIN {X 0,Y 93.403,Z 458.035,A -85,B 0,C 180,E1 -26920.842,E2 -26920.842} C_VEL
LIN {X 0,Y 96.018,Z 453.688,A -85,B 0,C 180,E1 -26927.024,E2 -26927.024} C_VEL
LIN {X 0,Y 99.538,Z 448.159,A -85,B 0,C 180,E1 -26932.851,E2 -26932.851} C_VEL
LIN {X 0,Y 103.983,Z 441.259,A -85,B 0,C 180,E1 -26938.237,E2 -26938.237} C_VEL
LIN {X 0,Y 109.017,Z 432.885,A -85,B 0,C 180,E1 -26943.041,E2 -26943.041} C_VEL
LIN {X 0,Y 114.043,Z 423.754,A -85,B 0,C 180,E1 -26946.931,E2 -26946.931} C_VEL
LIN {X 0,Y 118.739,Z 414.028,A -85,B 0,C 180,E1 -26950.066,E2 -26950.066} C_VEL
LIN {X 0,Y 123.181,Z 403.342,A -85,B 0,C 180,E1 -26952.65,E2 -26952.65} C_VEL
LIN {X 0,Y 127.226,Z 391.362,A -85,B 0,C 180,E1 -26954.774,E2 -26954.774} C_VEL
LIN {X 0,Y 130.296,Z 379.526,A -85,B 0,C 180,E1 -26956.313,E2 -26956.313} C_VEL
LIN {X 0,Y 132.647,Z 367.009,A -85,B 0,C 180,E1 -26957.431,E2 -26957.431} C_VEL
LIN {X 0,Y 134.274,Z 352.266,A -85,B 0,C 180,E1 -26958.179,E2 -26958.179} C_VEL
LIN {X 0,Y 136.339,Z 326.795,A -85,B 0,C 180,E1 -26959.214,E2 -26959.214} C_VEL
LIN {X 0,Y 132.419,Z 318.457,A -85,B 0,C 180,E1 -26962.262,E2 -26962.262} C_VEL
LIN {X 0,Y 128.272,Z 310.84,A -85,B 0,C 180,E1 -26965.869,E2 -26965.869} C_VEL
LIN {X 0,Y 124.188,Z 304.134,A -85,B 0,C 180,E1 -26970.019,E2 -26970.019} C_VEL
LIN {X 0,Y 121.624,Z 300.232,A -85,B 0,C 180,E1 -26973.086,E2 -26973.086} C_VEL
LIN {X 0,Y 119.033,Z 296.327,A -85,B 0,C 180,E1 -26976.777,E2 -26976.777} C_VEL
LIN {X 0,Y 116.672,Z 293.321,A -85,B 0,C 180,E1 -26980.906,E2 -26980.906} C_VEL
LIN {X 0,Y 115.845,Z 291.596,A -85,B 0,C 180,E1 -26982.845,E2 -26982.845} C_VEL
LIN {X 0,Y 113.668,Z 289.412,A -85,B 0,C 180,E1 -26989.31,E2 -26989.31} C_VEL
LIN {X 0,Y 112.996,Z 287.003,A -85,B 0,C 180,E1 -26996.434,E2 -26996.434} C_VEL
LIN {X 0,Y 113.129,Z 287.11,A -85,B 0,C 180,E1 -26999.777,E2 -26999.777} C_VEL
LIN {X 0,Y 114.267,Z 290.128,A -85,B 0,C 180,E1 -27006.622,E2 -27006.622} C_VEL
LIN {X 0,Y 116.033,Z 291.719,A -85,B 0,C 180,E1 -27011.203,E2 -27011.203} C_VEL
LIN {X 0,Y 117.959,Z 295.174,A -85,B 0,C 180,E1 -27015.164,E2 -27015.164} C_VEL
LIN {X 0,Y 119.472,Z 296.916,A -85,B 0,C 180,E1 -27017.539,E2 -27017.539} C_VEL
LIN {X 0,Y 122.629,Z 301.707,A -85,B 0,C 180,E1 -27021.813,E2 -27021.813} C_VEL
LIN {X 0,Y 125.689,Z 306.491,A -85,B 0,C 180,E1 -27025.236,E2 -27025.236} C_VEL
LIN {X 0,Y 129.412,Z 312.797,A -85,B 0,C 180,E1 -27028.814,E2 -27028.814} C_VEL
LIN {X 0,Y 131.485,Z 316.977,A -85,B 0,C 180,E1 -27030.645,E2 -27030.645} C_VEL
LIN {X 0,Y 134.681,Z 325.718,A -85,B 0,C 180,E1 -27033.407,E2 -27033.407} C_VEL
LIN {X 0,Y 136.103,Z 330.438,A -85,B 0,C 180,E1 -27034.611,E2 -27034.611} C_VEL
LIN {X 0,Y 133.003,Z 366.965,A -85,B 0,C 180,E1 -27036.167,E2 -27036.167} C_VEL
LIN {X 0,Y 130.817,Z 379.999,A -85,B 0,C 180,E1 -27037.112,E2 -27037.112} C_VEL
LIN {X 0,Y 127.799,Z 392.093,A -85,B 0,C 180,E1 -27038.405,E2 -27038.405} C_VEL
LIN {X 0,Y 124.114,Z 403.499,A -85,B 0,C 180,E1 -27040.143,E2 -27040.143} C_VEL
LIN {X 0,Y 119.415,Z 415.235,A -85,B 0,C 180,E1 -27042.636,E2 -27042.636} C_VEL
LIN {X 0,Y 114.388,Z 425.773,A -85,B 0,C 180,E1 -27045.663,E2 -27045.663} C_VEL
LIN {X 0,Y 109.739,Z 434.382,A -85,B 0,C 180,E1 -27048.971,E2 -27048.971} C_VEL
LIN {X 0,Y 105.171,Z 442.327,A -85,B 0,C 180,E1 -27053.028,E2 -27053.028} C_VEL
LIN {X 0,Y 100.514,Z 450.081,A -85,B 0,C 180,E1 -27058.372,E2 -27058.372} C_VEL
LIN {X 0,Y 96.557,Z 456.289,A -85,B 0,C 180,E1 -27064.106,E2 -27064.106} C_VEL
LIN {X 0,Y 93.609,Z 461.216,A -85,B 0,C 180,E1 -27070.254,E2 -27070.254} C_VEL
LIN {X 0,Y 91.843,Z 465.011,A -85,B 0,C 180,E1 -27076.729,E2 -27076.729} C_VEL
LIN {X 0,Y 91.169,Z 466.963,A -85,B 0,C 180,E1 -27081.131,E2 -27081.131} C_VEL
LIN {X 0,Y 90.921,Z 468.493,A -85,B 0,C 180,E1 -27085.567,E2 -27085.567} C_VEL
LIN {X 0,Y 90.978,Z 469.561,A -85,B 0,C 180,E1 -27090,E2 -27090} C_VEL
LIN {X 0,Y 90.929,Z 470.216,A -85,B 0,C 180,E1 -27094.433,E2 -27094.433} C_VEL
LIN {X 0,Y 91.213,Z 470.484,A -85,B 0,C 180,E1 -27098.865,E2 -27098.865} C_VEL
LIN {X 0,Y 91.886,Z 470.366,A -85,B 0,C 180,E1 -27103.265,E2 -27103.265} C_VEL
LIN {X 0,Y 94.703,Z 468.891,A -85,B 0,C 180,E1 -27111.781,E2 -27111.781} C_VEL
LIN {X 0,Y 99.57,Z 465.849,A -85,B 0,C 180,E1 -27119.61,E2 -27119.61} C_VEL
LIN {X 0,Y 104.303,Z 462.405,A -85,B 0,C 180,E1 -27124.941,E2 -27124.941} C_VEL
LIN {X 0,Y 110.008,Z 457.732,A -85,B 0,C 180,E1 -27129.948,E2 -27129.948} C_VEL
LIN {X 0,Y 117.073,Z 451.092,A -85,B 0,C 180,E1 -27134.859,E2 -27134.859} C_VEL
LIN {X 0,Y 124.057,Z 443.716,A -85,B 0,C 180,E1 -27138.645,E2 -27138.645} C_VEL
LIN {X 0,Y 131.614,Z 434.569,A -85,B 0,C 180,E1 -27141.965,E2 -27141.965} C_VEL
LIN {X 0,Y 138.859,Z 424.007,A -85,B 0,C 180,E1 -27144.699,E2 -27144.699} C_VEL
LIN {X 0,Y 145.083,Z 413.265,A -85,B 0,C 180,E1 -27146.679,E2 -27146.679} C_VEL
LIN {X 0,Y 150.019,Z 402.824,A -85,B 0,C 180,E1 -27148.117,E2 -27148.117} C_VEL
LIN {X 0,Y 154.628,Z 390.291,A -85,B 0,C 180,E1 -27149.398,E2 -27149.398} C_VEL
LIN {X 0,Y 158.24,Z 377.069,A -85,B 0,C 180,E1 -27150.321,E2 -27150.321} C_VEL
LIN {X 0,Y 158.888,Z 374.047,A -85,B 0,C 180,E1 -27150.459,E2 -27150.459} C_VEL
LIN {X 0,Y 159.626,Z 368.687,A -85,B 0,C 180,E1 -27150.873,E2 -27150.873} C_VEL
LIN {X 0,Y 159.7,Z 363.502,A -85,B 0,C 180,E1 -27151.561,E2 -27151.561} C_VEL
LIN {X 0,Y 159.151,Z 358.804,A -85,B 0,C 180,E1 -27152.535,E2 -27152.535} C_VEL
LIN {X 0,Y 158.042,Z 354.938,A -85,B 0,C 180,E1 -27153.848,E2 -27153.848} C_VEL
LIN {X 0,Y 155.591,Z 347.397,A -85,B 0,C 180,E1 -27156.983,E2 -27156.983} C_VEL
LIN {X 0,Y 153.496,Z 341.635,A -85,B 0,C 180,E1 -27160.091,E2 -27160.091} C_VEL
LIN {X 0,Y 151.223,Z 337.373,A -85,B 0,C 180,E1 -27163.982,E2 -27163.982} C_VEL
LIN {X 0,Y 149.738,Z 334.342,A -85,B 0,C 180,E1 -27167.463,E2 -27167.463} C_VEL
LIN {X 0,Y 148.249,Z 331.021,A -85,B 0,C 180,E1 -27173.706,E2 -27173.706} C_VEL
LIN {X 0,Y 148.199,Z 330.233,A -85,B 0,C 180,E1 -27174.795,E2 -27174.795} C_VEL
LIN {X 0,Y 148.195,Z 330.09,A -85,B 0,C 180,E1 -27179.433,E2 -27179.433} C_VEL
LIN {X 0,Y 149.978,Z 334.618,A -85,B 0,C 180,E1 -27187.552,E2 -27187.552} C_VEL
LIN {X 0,Y 151.996,Z 338.763,A -85,B 0,C 180,E1 -27191.883,E2 -27191.883} C_VEL
LIN {X 0,Y 154.044,Z 342.725,A -85,B 0,C 180,E1 -27195.145,E2 -27195.145} C_VEL
LIN {X 0,Y 156.579,Z 348.082,A -85,B 0,C 180,E1 -27198.482,E2 -27198.482} C_VEL
LIN {X 0,Y 158.652,Z 352.755,A -85,B 0,C 180,E1 -27200.841,E2 -27200.841} C_VEL
LIN {X 0,Y 156.809,Z 367.135,A -85,B 0,C 180,E1 -27201.374,E2 -27201.374} C_VEL
LIN {X 0,Y 153.91,Z 380.036,A -85,B 0,C 180,E1 -27202.171,E2 -27202.171} C_VEL
LIN {X 0,Y 150.052,Z 392.018,A -85,B 0,C 180,E1 -27203.194,E2 -27203.194} C_VEL
LIN {X 0,Y 144.975,Z 404.11,A -85,B 0,C 180,E1 -27204.639,E2 -27204.639} C_VEL
LIN {X 0,Y 139.202,Z 414.84,A -85,B 0,C 180,E1 -27206.342,E2 -27206.342} C_VEL
LIN {X 0,Y 132.469,Z 425.289,A -85,B 0,C 180,E1 -27208.662,E2 -27208.662} C_VEL
LIN {X 0,Y 125.606,Z 434.311,A -85,B 0,C 180,E1 -27211.43,E2 -27211.43} C_VEL
LIN {X 0,Y 117.857,Z 442.731,A -85,B 0,C 180,E1 -27214.921,E2 -27214.921} C_VEL
LIN {X 0,Y 110.745,Z 449.487,A -85,B 0,C 180,E1 -27218.977,E2 -27218.977} C_VEL
LIN {X 0,Y 103.242,Z 455.662,A -85,B 0,C 180,E1 -27224.375,E2 -27224.375} C_VEL
LIN {X 0,Y 97.539,Z 459.654,A -85,B 0,C 180,E1 -27229.573,E2 -27229.573} C_VEL
LIN {X 0,Y 94.252,Z 461.699,A -85,B 0,C 180,E1 -27233.378,E2 -27233.378} C_VEL
LIN {X 0,Y 90.705,Z 463.679,A -85,B 0,C 180,E1 -27238.464,E2 -27238.464} C_VEL
LIN {X 0,Y 86.851,Z 465.325,A -85,B 0,C 180,E1 -27246.134,E2 -27246.134} C_VEL
LIN {X 0,Y 84.298,Z 465.678,A -85,B 0,C 180,E1 -27255.516,E2 -27255.516} C_VEL
LIN {X 0,Y 83.818,Z 465.277,A -85,B 0,C 180,E1 -27260.346,E2 -27260.346} C_VEL
LIN {X 0,Y 83.762,Z 464.466,A -85,B 0,C 180,E1 -27265.187,E2 -27265.187} C_VEL
LIN {X 0,Y 84.513,Z 462.015,A -85,B 0,C 180,E1 -27273.696,E2 -27273.696} C_VEL
LIN {X 0,Y 86.446,Z 458.367,A -85,B 0,C 180,E1 -27281.727,E2 -27281.727} C_VEL
LIN {X 0,Y 89.264,Z 454.061,A -85,B 0,C 180,E1 -27288.356,E2 -27288.356} C_VEL
LIN {X 0,Y 93.046,Z 448.577,A -85,B 0,C 180,E1 -27294.546,E2 -27294.546} C_VEL
LIN {X 0,Y 97.796,Z 441.731,A -85,B 0,C 180,E1 -27300.202,E2 -27300.202} C_VEL
LIN {X 0,Y 102.894,Z 433.894,A -85,B 0,C 180,E1 -27304.95,E2 -27304.95} C_VEL
LIN {X 0,Y 108.468,Z 424.377,A -85,B 0,C 180,E1 -27309.178,E2 -27309.178} C_VEL
LIN {X 0,Y 113.993,Z 413.567,A -85,B 0,C 180,E1 -27312.701,E2 -27312.701} C_VEL
LIN {X 0,Y 118.674,Z 402.659,A -85,B 0,C 180,E1 -27315.288,E2 -27315.288} C_VEL
LIN {X 0,Y 122.934,Z 390.446,A -85,B 0,C 180,E1 -27317.396,E2 -27317.396} C_VEL
LIN {X 0,Y 126.143,Z 378.415,A -85,B 0,C 180,E1 -27318.892,E2 -27318.892} C_VEL
LIN {X 0,Y 128.513,Z 365.627,A -85,B 0,C 180,E1 -27319.962,E2 -27319.962} C_VEL
LIN {X 0,Y 130.318,Z 348.512,A -85,B 0,C 180,E1 -27320.764,E2 -27320.764} C_VEL
LIN {X 0,Y 131.909,Z 329.53,A -85,B 0,C 180,E1 -27321.546,E2 -27321.546} C_VEL
LIN {X 0,Y 128.356,Z 321.857,A -85,B 0,C 180,E1 -27324.648,E2 -27324.648} C_VEL
LIN {X 0,Y 124.109,Z 313.858,A -85,B 0,C 180,E1 -27328.886,E2 -27328.886} C_VEL
LIN {X 0,Y 120.838,Z 308.48,A -85,B 0,C 180,E1 -27332.74,E2 -27332.74} C_VEL
LIN {X 0,Y 119.41,Z 306.222,A -85,B 0,C 180,E1 -27334.678,E2 -27334.678} C_VEL
LIN {X 0,Y 117.257,Z 302.782,A -85,B 0,C 180,E1 -27338.068,E2 -27338.068} C_VEL
LIN {X 0,Y 115.016,Z 299.459,A -85,B 0,C 180,E1 -27342.512,E2 -27342.512} C_VEL
LIN {X 0,Y 114.461,Z 298.408,A -85,B 0,C 180,E1 -27343.935,E2 -27343.935} C_VEL
LIN {X 0,Y 112.115,Z 294.172,A -85,B 0,C 180,E1 -27356.406,E2 -27356.406} C_VEL
LIN {X 0,Y 112.219,Z 294.162,A -85,B 0,C 180,E1 -27359.327,E2 -27359.327} C_VEL
LIN {X 0,Y 113.242,Z 297.077,A -85,B 0,C 180,E1 -27366.145,E2 -27366.145} C_VEL
LIN {X 0,Y 114.74,Z 298.62,A -85,B 0,C 180,E1 -27370.365,E2 -27370.365} C_VEL
LIN {X 0,Y 116.78,Z 302.209,A -85,B 0,C 180,E1 -27374.763,E2 -27374.763} C_VEL
LIN {X 0,Y 117.791,Z 303.52,A -85,B 0,C 180,E1 -27376.464,E2 -27376.464} C_VEL
LIN {X 0,Y 120.52,Z 307.885,A -85,B 0,C 180,E1 -27380.48,E2 -27380.48} C_VEL
LIN {X 0,Y 124.045,Z 313.637,A -85,B 0,C 180,E1 -27384.677,E2 -27384.677} C_VEL
LIN {X 0,Y 127.838,Z 320.93,A -85,B 0,C 180,E1 -27388.528,E2 -27388.528} C_VEL
LIN {X 0,Y 130.755,Z 329.329,A -85,B 0,C 180,E1 -27391.357,E2 -27391.357} C_VEL
LIN {X 0,Y 131.699,Z 332.556,A -85,B 0,C 180,E1 -27392.252,E2 -27392.252} C_VEL
LIN {X 0,Y 128.589,Z 367.248,A -85,B 0,C 180,E1 -27393.741,E2 -27393.741} C_VEL
LIN {X 0,Y 126.115,Z 380.861,A -85,B 0,C 180,E1 -27394.718,E2 -27394.718} C_VEL
LIN {X 0,Y 122.868,Z 393.209,A -85,B 0,C 180,E1 -27396.104,E2 -27396.104} C_VEL
LIN {X 0,Y 118.368,Z 405.85,A -85,B 0,C 180,E1 -27398.122,E2 -27398.122} C_VEL
LIN {X 0,Y 113.493,Z 417.118,A -85,B 0,C 180,E1 -27400.662,E2 -27400.662} C_VEL
LIN {X 0,Y 108.83,Z 426.222,A -85,B 0,C 180,E1 -27403.407,E2 -27403.407} C_VEL
LIN {X 0,Y 103.431,Z 435.557,A -85,B 0,C 180,E1 -27407.197,E2 -27407.197} C_VEL
LIN {X 0,Y 98.02,Z 444.209,A -85,B 0,C 180,E1 -27412.064,E2 -27412.064} C_VEL
LIN {X 0,Y 94.535,Z 449.661,A -85,B 0,C 180,E1 -27416.112,E2 -27416.112} C_VEL
LIN {X 0,Y 90.199,Z 455.911,A -85,B 0,C 180,E1 -27422.128,E2 -27422.128} C_VEL
LIN {X 0,Y 86.924,Z 460.875,A -85,B 0,C 180,E1 -27428.664,E2 -27428.664} C_VEL
LIN {X 0,Y 84.927,Z 464.707,A -85,B 0,C 180,E1 -27435.626,E2 -27435.626} C_VEL
LIN {X 0,Y 84.148,Z 466.677,A -85,B 0,C 180,E1 -27440.384,E2 -27440.384} C_VEL
LIN {X 0,Y 83.825,Z 468.228,A -85,B 0,C 180,E1 -27445.191,E2 -27445.191} C_VEL
LIN {X 0,Y 83.884,Z 469.325,A -85,B 0,C 180,E1 -27450,E2 -27450} C_VEL
LIN {X 0,Y 83.862,Z 469.996,A -85,B 0,C 180,E1 -27454.807,E2 -27454.807} C_VEL
LIN {X 0,Y 84.185,Z 470.278,A -85,B 0,C 180,E1 -27459.612,E2 -27459.612} C_VEL
LIN {X 0,Y 84.976,Z 470.179,A -85,B 0,C 180,E1 -27464.366,E2 -27464.366} C_VEL
LIN {X 0,Y 86.3,Z 469.67,A -85,B 0,C 180,E1 -27469.011,E2 -27469.011} C_VEL
LIN {X 0,Y 90.535,Z 467.445,A -85,B 0,C 180,E1 -27477.76,E2 -27477.76} C_VEL
LIN {X 0,Y 95.024,Z 464.701,A -85,B 0,C 180,E1 -27483.69,E2 -27483.69} C_VEL
LIN {X 0,Y 100.471,Z 460.953,A -85,B 0,C 180,E1 -27489.018,E2 -27489.018} C_VEL
LIN {X 0,Y 106.566,Z 456.101,A -85,B 0,C 180,E1 -27493.826,E2 -27493.826} C_VEL
LIN {X 0,Y 113.324,Z 450.004,A -85,B 0,C 180,E1 -27498.091,E2 -27498.091} C_VEL
LIN {X 0,Y 120.772,Z 442.439,A -85,B 0,C 180,E1 -27501.776,E2 -27501.776} C_VEL
LIN {X 0,Y 127.369,Z 434.718,A -85,B 0,C 180,E1 -27504.477,E2 -27504.477} C_VEL
LIN {X 0,Y 134.88,Z 424.244,A -85,B 0,C 180,E1 -27507.162,E2 -27507.162} C_VEL
LIN {X 0,Y 141.318,Z 413.591,A -85,B 0,C 180,E1 -27509.079,E2 -27509.079} C_VEL
LIN {X 0,Y 146.408,Z 403.296,A -85,B 0,C 180,E1 -27510.465,E2 -27510.465} C_VEL
LIN {X 0,Y 151.158,Z 391.007,A -85,B 0,C 180,E1 -27511.702,E2 -27511.702} C_VEL
LIN {X 0,Y 154.906,Z 377.927,A -85,B 0,C 180,E1 -27512.604,E2 -27512.604} C_VEL
LIN {X 0,Y 157.41,Z 365.076,A -85,B 0,C 180,E1 -27513.135,E2 -27513.135} C_VEL
LIN {X 0,Y 158.355,Z 355.959,A -85,B 0,C 180,E1 -27513.476,E2 -27513.476} C_VEL
LIN {X 0,Y 158.042,Z 354.938,A -85,B 0,C 180,E1 -27513.848,E2 -27513.848} C_VEL
LIN {X 0,Y 156.44,Z 351.873,A -85,B 0,C 180,E1 -27515.61,E2 -27515.61} C_VEL
LIN {X 0,Y 154.742,Z 349.633,A -85,B 0,C 180,E1 -27517.55,E2 -27517.55} C_VEL
LIN {X 0,Y 149.972,Z 344.168,A -85,B 0,C 180,E1 -27524.634,E2 -27524.634} C_VEL
LIN {X 0,Y 148.504,Z 341.048,A -85,B 0,C 180,E1 -27528.397,E2 -27528.397} C_VEL
LIN {X 0,Y 147.306,Z 337.747,A -85,B 0,C 180,E1 -27534.525,E2 -27534.525} C_VEL
LIN {X 0,Y 147.257,Z 337.127,A -85,B 0,C 180,E1 -27535.894,E2 -27535.894} C_VEL
LIN {X 0,Y 147.32,Z 337.318,A -85,B 0,C 180,E1 -27539.572,E2 -27539.572} C_VEL
LIN {X 0,Y 148.811,Z 341.428,A -85,B 0,C 180,E1 -27546.866,E2 -27546.866} C_VEL
LIN {X 0,Y 150.621,Z 345.433,A -85,B 0,C 180,E1 -27551.097,E2 -27551.097} C_VEL
LIN {X 0,Y 152.772,Z 349.897,A -85,B 0,C 180,E1 -27554.742,E2 -27554.742} C_VEL
LIN {X 0,Y 155.533,Z 356.355,A -85,B 0,C 180,E1 -27558.525,E2 -27558.525} C_VEL
LIN {X 0,Y 153.758,Z 368.65,A -85,B 0,C 180,E1 -27559.047,E2 -27559.047} C_VEL
LIN {X 0,Y 150.644,Z 381.601,A -85,B 0,C 180,E1 -27559.849,E2 -27559.849} C_VEL
LIN {X 0,Y 146.625,Z 393.35,A -85,B 0,C 180,E1 -27560.825,E2 -27560.825} C_VEL
LIN {X 0,Y 141.398,Z 405.13,A -85,B 0,C 180,E1 -27562.22,E2 -27562.22} C_VEL
LIN {X 0,Y 134.705,Z 416.887,A -85,B 0,C 180,E1 -27564.072,E2 -27564.072} C_VEL
LIN {X 0,Y 128.608,Z 425.852,A -85,B 0,C 180,E1 -27566.065,E2 -27566.065} C_VEL
LIN {X 0,Y 122.031,Z 434.155,A -85,B 0,C 180,E1 -27568.564,E2 -27568.564} C_VEL
LIN {X 0,Y 115.228,Z 441.38,A -85,B 0,C 180,E1 -27571.363,E2 -27571.363} C_VEL
LIN {X 0,Y 107.575,Z 448.454,A -85,B 0,C 180,E1 -27575.25,E2 -27575.25} C_VEL
LIN {X 0,Y 100.53,Z 454.077,A -85,B 0,C 180,E1 -27579.735,E2 -27579.735} C_VEL
LIN {X 0,Y 94.13,Z 458.484,A -85,B 0,C 180,E1 -27584.822,E2 -27584.822} C_VEL
LIN {X 0,Y 88.567,Z 461.801,A -85,B 0,C 180,E1 -27590.593,E2 -27590.593} C_VEL
LIN {X 0,Y 82.638,Z 464.671,A -85,B 0,C 180,E1 -27599.318,E2 -27599.318} C_VEL
LIN {X 0,Y 80.336,Z 465.496,A -85,B 0,C 180,E1 -27604.061,E2 -27604.061} C_VEL
LIN {X 0,Y 77.383,Z 465.885,A -85,B 0,C 180,E1 -27614.189,E2 -27614.189} C_VEL
LIN {X 0,Y 76.758,Z 465.502,A -85,B 0,C 180,E1 -27619.448,E2 -27619.448} C_VEL
LIN {X 0,Y 76.642,Z 464.724,A -85,B 0,C 180,E1 -27624.738,E2 -27624.738} C_VEL
LIN {X 0,Y 76.912,Z 463.513,A -85,B 0,C 180,E1 -27630,E2 -27630} C_VEL
LIN {X 0,Y 78.122,Z 460.959,A -85,B 0,C 180,E1 -27637.755,E2 -27637.755} C_VEL
LIN {X 0,Y 80.42,Z 457.413,A -85,B 0,C 180,E1 -27645.199,E2 -27645.199} C_VEL
LIN {X 0,Y 83.839,Z 452.767,A -85,B 0,C 180,E1 -27652.162,E2 -27652.162} C_VEL
LIN {X 0,Y 89.068,Z 445.777,A -85,B 0,C 180,E1 -27659.548,E2 -27659.548} C_VEL
LIN {X 0,Y 94.605,Z 438.202,A -85,B 0,C 180,E1 -27665.15,E2 -27665.15} C_VEL
LIN {X 0,Y 99.731,Z 430.455,A -85,B 0,C 180,E1 -27669.362,E2 -27669.362} C_VEL
LIN {X 0,Y 105.956,Z 419.924,A -85,B 0,C 180,E1 -27673.485,E2 -27673.485} C_VEL
LIN {X 0,Y 111.345,Z 409.209,A -85,B 0,C 180,E1 -27676.541,E2 -27676.541} C_VEL
LIN {X 0,Y 115.698,Z 398.792,A -85,B 0,C 180,E1 -27678.739,E2 -27678.739} C_VEL
LIN {X 0,Y 119.779,Z 386.498,A -85,B 0,C 180,E1 -27680.627,E2 -27680.627} C_VEL
LIN {X 0,Y 122.978,Z 373.644,A -85,B 0,C 180,E1 -27681.991,E2 -27681.991} C_VEL
LIN {X 0,Y 124.979,Z 361.549,A -85,B 0,C 180,E1 -27682.837,E2 -27682.837} C_VEL
LIN {X 0,Y 127.693,Z 332.439,A -85,B 0,C 180,E1 -27684.028,E2 -27684.028} C_VEL
LIN {X 0,Y 124.135,Z 324.603,A -85,B 0,C 180,E1 -27687.585,E2 -27687.585} C_VEL
LIN {X 0,Y 120.755,Z 318.172,A -85,B 0,C 180,E1 -27691.47,E2 -27691.47} C_VEL
LIN {X 0,Y 117.858,Z 312.963,A -85,B 0,C 180,E1 -27695.479,E2 -27695.479} C_VEL
LIN {X 0,Y 115.642,Z 309.327,A -85,B 0,C 180,E1 -27699.221,E2 -27699.221} C_VEL
LIN {X 0,Y 113.524,Z 305.781,A -85,B 0,C 180,E1 -27703.951,E2 -27703.951} C_VEL
LIN {X 0,Y 113.08,Z 305.169,A -85,B 0,C 180,E1 -27705.167,E2 -27705.167} C_VEL
LIN {X 0,Y 111.241,Z 301.284,A -85,B 0,C 180,E1 -27716.377,E2 -27716.377} C_VEL
LIN {X 0,Y 111.313,Z 301.12,A -85,B 0,C 180,E1 -27718.643,E2 -27718.643} C_VEL
LIN {X 0,Y 112.37,Z 304.189,A -85,B 0,C 180,E1 -27726.193,E2 -27726.193} C_VEL
LIN {X 0,Y 113.461,Z 305.476,A -85,B 0,C 180,E1 -27729.47,E2 -27729.47} C_VEL
LIN {X 0,Y 115.467,Z 309.046,A -85,B 0,C 180,E1 -27734.091,E2 -27734.091} C_VEL
LIN {X 0,Y 116.438,Z 310.693,A -85,B 0,C 180,E1 -27735.879,E2 -27735.879} C_VEL
LIN {X 0,Y 118.697,Z 314.475,A -85,B 0,C 180,E1 -27739.419,E2 -27739.419} C_VEL
LIN {X 0,Y 121.627,Z 319.581,A -85,B 0,C 180,E1 -27743.217,E2 -27743.217} C_VEL
LIN {X 0,Y 124.805,Z 326.07,A -85,B 0,C 180,E1 -27746.775,E2 -27746.775} C_VEL
LIN {X 0,Y 127.445,Z 334.382,A -85,B 0,C 180,E1 -27749.642,E2 -27749.642} C_VEL
LIN {X 0,Y 127.196,Z 338.999,A -85,B 0,C 180,E1 -27749.939,E2 -27749.939} C_VEL
LIN {X 0,Y 124.475,Z 367.083,A -85,B 0,C 180,E1 -27751.116,E2 -27751.116} C_VEL
LIN {X 0,Y 122.05,Z 380.197,A -85,B 0,C 180,E1 -27752.054,E2 -27752.054} C_VEL
LIN {X 0,Y 118.79,Z 392.141,A -85,B 0,C 180,E1 -27753.313,E2 -27753.313} C_VEL
LIN {X 0,Y 114.791,Z 403.423,A -85,B 0,C 180,E1 -27755.028,E2 -27755.028} C_VEL
LIN {X 0,Y 109.609,Z 415.094,A -85,B 0,C 180,E1 -27757.489,E2 -27757.489} C_VEL
LIN {X 0,Y 104.064,Z 425.591,A -85,B 0,C 180,E1 -27760.556,E2 -27760.556} C_VEL
LIN {X 0,Y 98.303,Z 435.027,A -85,B 0,C 180,E1 -27764.363,E2 -27764.363} C_VEL
LIN {X 0,Y 92.036,Z 444.387,A -85,B 0,C 180,E1 -27769.783,E2 -27769.783} C_VEL
LIN {X 0,Y 87.819,Z 450.362,A -85,B 0,C 180,E1 -27774.535,E2 -27774.535} C_VEL
LIN {X 0,Y 82.608,Z 457.354,A -85,B 0,C 180,E1 -27782.101,E2 -27782.101} C_VEL
LIN {X 0,Y 79.429,Z 461.969,A -85,B 0,C 180,E1 -27789.272,E2 -27789.272} C_VEL
LIN {X 0,Y 78.027,Z 464.402,A -85,B 0,C 180,E1 -27794.323,E2 -27794.323} C_VEL
LIN {X 0,Y 77.13,Z 466.39,A -85,B 0,C 180,E1 -27799.5,E2 -27799.5} C_VEL
LIN {X 0,Y 76.753,Z 467.96,A -85,B 0,C 180,E1 -27804.746,E2 -27804.746} C_VEL
LIN {X 0,Y 76.782,Z 469.088,A -85,B 0,C 180,E1 -27810,E2 -27810} C_VEL
LIN {X 0,Y 76.782,Z 469.775,A -85,B 0,C 180,E1 -27815.252,E2 -27815.252} C_VEL
LIN {X 0,Y 77.189,Z 470.074,A -85,B 0,C 180,E1 -27820.492,E2 -27820.492} C_VEL
LIN {X 0,Y 79.602,Z 469.512,A -85,B 0,C 180,E1 -27830.681,E2 -27830.681} C_VEL
LIN {X 0,Y 81.624,Z 468.609,A -85,B 0,C 180,E1 -27835.5,E2 -27835.5} C_VEL
LIN {X 0,Y 87.475,Z 465.636,A -85,B 0,C 180,E1 -27844.222,E2 -27844.222} C_VEL
LIN {X 0,Y 93.012,Z 462.262,A -85,B 0,C 180,E1 -27849.961,E2 -27849.961} C_VEL
LIN {X 0,Y 99.29,Z 457.83,A -85,B 0,C 180,E1 -27855.059,E2 -27855.059} C_VEL
LIN {X 0,Y 107.457,Z 451.15,A -85,B 0,C 180,E1 -27860.218,E2 -27860.218} C_VEL
LIN {X 0,Y 115.166,Z 443.871,A -85,B 0,C 180,E1 -27863.958,E2 -27863.958} C_VEL
LIN {X 0,Y 123.386,Z 434.855,A -85,B 0,C 180,E1 -27867.157,E2 -27867.157} C_VEL
LIN {X 0,Y 130.421,Z 425.55,A -85,B 0,C 180,E1 -27869.564,E2 -27869.564} C_VEL
LIN {X 0,Y 137.073,Z 415.206,A -85,B 0,C 180,E1 -27871.406,E2 -27871.406} C_VEL
LIN {X 0,Y 143.056,Z 403.739,A -85,B 0,C 180,E1 -27872.929,E2 -27872.929} C_VEL
LIN {X 0,Y 147.944,Z 391.723,A -85,B 0,C 180,E1 -27874.108,E2 -27874.108} C_VEL
LIN {X 0,Y 151.87,Z 378.624,A -85,B 0,C 180,E1 -27874.991,E2 -27874.991} C_VEL
LIN {X 0,Y 154.587,Z 365.407,A -85,B 0,C 180,E1 -27875.516,E2 -27875.516} C_VEL
LIN {X 0,Y 155.337,Z 359.131,A -85,B 0,C 180,E1 -27875.74,E2 -27875.74} C_VEL
LIN {X 0,Y 153.063,Z 351.54,A -85,B 0,C 180,E1 -27879.099,E2 -27879.099} C_VEL
LIN {X 0,Y 151.676,Z 347.598,A -85,B 0,C 180,E1 -27881.429,E2 -27881.429} C_VEL
LIN {X 0,Y 149.972,Z 344.168,A -85,B 0,C 180,E1 -27884.634,E2 -27884.634} C_VEL
LIN {X 0,Y 149.232,Z 343.631,A -85,B 0,C 180,E1 -27886.104,E2 -27886.104} C_VEL
LIN {X 0,Y 147.956,Z 344.789,A -85,B 0,C 180,E1 -27888.605,E2 -27888.605} C_VEL
LIN {X 0,Y 146.925,Z 346.222,A -85,B 0,C 180,E1 -27891.167,E2 -27891.167} C_VEL
LIN {X 0,Y 146.571,Z 346.076,A -85,B 0,C 180,E1 -27892.733,E2 -27892.733} C_VEL
LIN {X 0,Y 146.387,Z 344.212,A -85,B 0,C 180,E1 -27895.871,E2 -27895.871} C_VEL
LIN {X 0,Y 146.421,Z 344.283,A -85,B 0,C 180,E1 -27899.141,E2 -27899.141} C_VEL
LIN {X 0,Y 147.661,Z 348.213,A -85,B 0,C 180,E1 -27906.148,E2 -27906.148} C_VEL
LIN {X 0,Y 149.208,Z 351.913,A -85,B 0,C 180,E1 -27910.149,E2 -27910.149} C_VEL
LIN {X 0,Y 151.215,Z 356.443,A -85,B 0,C 180,E1 -27913.866,E2 -27913.866} C_VEL
LIN {X 0,Y 152.634,Z 360.283,A -85,B 0,C 180,E1 -27916.209,E2 -27916.209} C_VEL
LIN {X 0,Y 150.169,Z 373.757,A -85,B 0,C 180,E1 -27916.794,E2 -27916.794} C_VEL
LIN {X 0,Y 146.573,Z 386.316,A -85,B 0,C 180,E1 -27917.639,E2 -27917.639} C_VEL
LIN {X 0,Y 141.909,Z 398.217,A -85,B 0,C 180,E1 -27918.709,E2 -27918.709} C_VEL
LIN {X 0,Y 136.55,Z 409.01,A -85,B 0,C 180,E1 -27920.066,E2 -27920.066} C_VEL
LIN {X 0,Y 130.436,Z 418.895,A -85,B 0,C 180,E1 -27921.651,E2 -27921.651} C_VEL
LIN {X 0,Y 123.075,Z 428.893,A -85,B 0,C 180,E1 -27923.985,E2 -27923.985} C_VEL
LIN {X 0,Y 115.871,Z 437.064,A -85,B 0,C 180,E1 -27926.537,E2 -27926.537} C_VEL
LIN {X 0,Y 107.554,Z 445.06,A -85,B 0,C 180,E1 -27930.025,E2 -27930.025} C_VEL
LIN {X 0,Y 99.066,Z 451.951,A -85,B 0,C 180,E1 -27934.579,E2 -27934.579} C_VEL
LIN {X 0,Y 91.446,Z 457.178,A -85,B 0,C 180,E1 -27939.777,E2 -27939.777} C_VEL
LIN {X 0,Y 85.045,Z 460.886,A -85,B 0,C 180,E1 -27945.377,E2 -27945.377} C_VEL
LIN {X 0,Y 77.893,Z 464.29,A -85,B 0,C 180,E1 -27954.297,E2 -27954.297} C_VEL
LIN {X 0,Y 73.936,Z 465.661,A -85,B 0,C 180,E1 -27961.623,E2 -27961.623} C_VEL
LIN {X 0,Y 70.506,Z 466.092,A -85,B 0,C 180,E1 -27972.6,E2 -27972.6} C_VEL
LIN {X 0,Y 69.734,Z 465.726,A -85,B 0,C 180,E1 -27978.371,E2 -27978.371} C_VEL
LIN {X 0,Y 69.538,Z 464.975,A -85,B 0,C 180,E1 -27984.199,E2 -27984.199} C_VEL
LIN {X 0,Y 69.79,Z 463.789,A -85,B 0,C 180,E1 -27990,E2 -27990} C_VEL
LIN {X 0,Y 70.85,Z 461.711,A -85,B 0,C 180,E1 -27997.264,E2 -27997.264} C_VEL
LIN {X 0,Y 73.607,Z 457.763,A -85,B 0,C 180,E1 -28006.645,E2 -28006.645} C_VEL
LIN {X 0,Y 77.319,Z 453.16,A -85,B 0,C 180,E1 -28014.144,E2 -28014.144} C_VEL
LIN {X 0,Y 82.999,Z 446.213,A -85,B 0,C 180,E1 -28021.953,E2 -28021.953} C_VEL
LIN {X 0,Y 88.916,Z 438.696,A -85,B 0,C 180,E1 -28027.775,E2 -28027.775} C_VEL
LIN {X 0,Y 94.366,Z 431.019,A -85,B 0,C 180,E1 -28032.089,E2 -28032.089} C_VEL
LIN {X 0,Y 100.938,Z 420.582,A -85,B 0,C 180,E1 -28036.251,E2 -28036.251} C_VEL
LIN {X 0,Y 106.602,Z 409.964,A -85,B 0,C 180,E1 -28039.302,E2 -28039.302} C_VEL
LIN {X 0,Y 111.177,Z 399.695,A -85,B 0,C 180,E1 -28041.469,E2 -28041.469} C_VEL
LIN {X 0,Y 115.442,Z 387.668,A -85,B 0,C 180,E1 -28043.328,E2 -28043.328} C_VEL
LIN {X 0,Y 118.933,Z 374.456,A -85,B 0,C 180,E1 -28044.726,E2 -28044.726} C_VEL
LIN {X 0,Y 121.184,Z 361.515,A -85,B 0,C 180,E1 -28045.623,E2 -28045.623} C_VEL
LIN {X 0,Y 123.733,Z 335.35,A -85,B 0,C 180,E1 -28046.675,E2 -28046.675} C_VEL
LIN {X 0,Y 120.323,Z 327.689,A -85,B 0,C 180,E1 -28050.614,E2 -28050.614} C_VEL
LIN {X 0,Y 117.108,Z 321.389,A -85,B 0,C 180,E1 -28055.029,E2 -28055.029} C_VEL
LIN {X 0,Y 114.966,Z 317.497,A -85,B 0,C 180,E1 -28058.635,E2 -28058.635} C_VEL
LIN {X 0,Y 114.053,Z 315.847,A -85,B 0,C 180,E1 -28060.449,E2 -28060.449} C_VEL
LIN {X 0,Y 112.08,Z 312.162,A -85,B 0,C 180,E1 -28065.473,E2 -28065.473} C_VEL
LIN {X 0,Y 110.365,Z 308.412,A -85,B 0,C 180,E1 -28076.349,E2 -28076.349} C_VEL
LIN {X 0,Y 110.421,Z 308.616,A -85,B 0,C 180,E1 -28079.088,E2 -28079.088} C_VEL
LIN {X 0,Y 112.197,Z 312.285,A -85,B 0,C 180,E1 -28088.509,E2 -28088.509} C_VEL
LIN {X 0,Y 114.607,Z 316.794,A -85,B 0,C 180,E1 -28094.312,E2 -28094.312} C_VEL
LIN {X 0,Y 116.892,Z 321.001,A -85,B 0,C 180,E1 -28098.286,E2 -28098.286} C_VEL
LIN {X 0,Y 119.304,Z 325.548,A -85,B 0,C 180,E1 -28101.717,E2 -28101.717} C_VEL
LIN {X 0,Y 121.892,Z 331.235,A -85,B 0,C 180,E1 -28104.937,E2 -28104.937} C_VEL
LIN {X 0,Y 123.597,Z 337.074,A -85,B 0,C 180,E1 -28107.058,E2 -28107.058} C_VEL
LIN {X 0,Y 120.832,Z 365.726,A -85,B 0,C 180,E1 -28108.259,E2 -28108.259} C_VEL
LIN {X 0,Y 118.415,Z 378.898,A -85,B 0,C 180,E1 -28109.162,E2 -28109.162} C_VEL
LIN {X 0,Y 115.597,Z 389.161,A -85,B 0,C 180,E1 -28110.119,E2 -28110.119} C_VEL
LIN {X 0,Y 111.548,Z 400.791,A -85,B 0,C 180,E1 -28111.728,E2 -28111.728} C_VEL
LIN {X 0,Y 106.767,Z 411.693,A -85,B 0,C 180,E1 -28113.794,E2 -28113.794} C_VEL
LIN {X 0,Y 100.837,Z 422.802,A -85,B 0,C 180,E1 -28116.725,E2 -28116.725} C_VEL
LIN {X 0,Y 94.623,Z 432.705,A -85,B 0,C 180,E1 -28120.421,E2 -28120.421} C_VEL
LIN {X 0,Y 88.992,Z 440.831,A -85,B 0,C 180,E1 -28124.704,E2 -28124.704} C_VEL
LIN {X 0,Y 83.095,Z 448.809,A -85,B 0,C 180,E1 -28130.63,E2 -28130.63} C_VEL
LIN {X 0,Y 77.888,Z 455.15,A -85,B 0,C 180,E1 -28137.222,E2 -28137.222} C_VEL
LIN {X 0,Y 73.789,Z 460.19,A -85,B 0,C 180,E1 -28144.622,E2 -28144.622} C_VEL
LIN {X 0,Y 71.186,Z 464.096,A -85,B 0,C 180,E1 -28152.772,E2 -28152.772} C_VEL
LIN {X 0,Y 70.147,Z 466.103,A -85,B 0,C 180,E1 -28158.441,E2 -28158.441} C_VEL
LIN {X 0,Y 69.663,Z 467.689,A -85,B 0,C 180,E1 -28164.21,E2 -28164.21} C_VEL
LIN {X 0,Y 69.702,Z 468.851,A -85,B 0,C 180,E1 -28170,E2 -28170} C_VEL
LIN {X 0,Y 69.725,Z 469.554,A -85,B 0,C 180,E1 -28175.785,E2 -28175.785} C_VEL
LIN {X 0,Y 71.26,Z 469.801,A -85,B 0,C 180,E1 -28187.21,E2 -28187.21} C_VEL
LIN {X 0,Y 72.971,Z 469.349,A -85,B 0,C 180,E1 -28192.66,E2 -28192.66} C_VEL
LIN {X 0,Y 75.251,Z 468.469,A -85,B 0,C 180,E1 -28197.838,E2 -28197.838} C_VEL
LIN {X 0,Y 81.667,Z 465.529,A -85,B 0,C 180,E1 -28207.042,E2 -28207.042} C_VEL
LIN {X 0,Y 87.685,Z 462.191,A -85,B 0,C 180,E1 -28212.944,E2 -28212.944} C_VEL
LIN {X 0,Y 94.39,Z 457.797,A -85,B 0,C 180,E1 -28218.123,E2 -28218.123} C_VEL
LIN {X 0,Y 101.763,Z 452.227,A -85,B 0,C 180,E1 -28222.581,E2 -28222.581} C_VEL
LIN {X 0,Y 109.762,Z 445.291,A -85,B 0,C 180,E1 -28226.344,E2 -28226.344} C_VEL
LIN {X 0,Y 118.251,Z 436.613,A -85,B 0,C 180,E1 -28229.517,E2 -28229.517} C_VEL
LIN {X 0,Y 125.498,Z 427.743,A -85,B 0,C 180,E1 -28231.886,E2 -28231.886} C_VEL
LIN {X 0,Y 133.054,Z 416.815,A -85,B 0,C 180,E1 -28233.89,E2 -28233.89} C_VEL
LIN {X 0,Y 139.202,Z 405.761,A -85,B 0,C 180,E1 -28235.338,E2 -28235.338} C_VEL
LIN {X 0,Y 144.614,Z 393.389,A -85,B 0,C 180,E1 -28236.534,E2 -28236.534} C_VEL
LIN {X 0,Y 148.618,Z 381.268,A -85,B 0,C 180,E1 -28237.354,E2 -28237.354} C_VEL
LIN {X 0,Y 151.507,Z 368.809,A -85,B 0,C 180,E1 -28237.87,E2 -28237.87} C_VEL
LIN {X 0,Y 152.434,Z 362.241,A -85,B 0,C 180,E1 -28238.179,E2 -28238.179} C_VEL
LIN {X 0,Y 150.758,Z 356.001,A -85,B 0,C 180,E1 -28241.222,E2 -28241.222} C_VEL
LIN {X 0,Y 150.029,Z 353.801,A -85,B 0,C 180,E1 -28242.625,E2 -28242.625} C_VEL
LIN {X 0,Y 148.526,Z 350.561,A -85,B 0,C 180,E1 -28245.791,E2 -28245.791} C_VEL
LIN {X 0,Y 147.416,Z 347.893,A -85,B 0,C 180,E1 -28249.007,E2 -28249.007} C_VEL
LIN {X 0,Y 146.571,Z 346.076,A -85,B 0,C 180,E1 -28252.733,E2 -28252.733} C_VEL
LIN {X 0,Y 146.322,Z 346.029,A -85,B 0,C 180,E1 -28254.256,E2 -28254.256} C_VEL
LIN {X 0,Y 145.959,Z 347.548,A -85,B 0,C 180,E1 -28256.238,E2 -28256.238} C_VEL
LIN {X 0,Y 145.586,Z 352.023,A -85,B 0,C 180,E1 -28260.187,E2 -28260.187} C_VEL
LIN {X 0,Y 145.617,Z 352.386,A -85,B 0,C 180,E1 -28260.71,E2 -28260.71} C_VEL
LIN {X 0,Y 146.557,Z 355.062,A -85,B 0,C 180,E1 -28265.504,E2 -28265.504} C_VEL
LIN {X 0,Y 147.828,Z 358.462,A -85,B 0,C 180,E1 -28269.234,E2 -28269.234} C_VEL
LIN {X 0,Y 149.443,Z 362.791,A -85,B 0,C 180,E1 -28272.822,E2 -28272.822} C_VEL
LIN {X 0,Y 149.88,Z 364.214,A -85,B 0,C 180,E1 -28273.785,E2 -28273.785} C_VEL
LIN {X 0,Y 146.972,Z 377.632,A -85,B 0,C 180,E1 -28274.42,E2 -28274.42} C_VEL
LIN {X 0,Y 142.848,Z 390.321,A -85,B 0,C 180,E1 -28275.288,E2 -28275.288} C_VEL
LIN {X 0,Y 137.401,Z 402.653,A -85,B 0,C 180,E1 -28276.452,E2 -28276.452} C_VEL
LIN {X 0,Y 131.088,Z 413.875,A -85,B 0,C 180,E1 -28277.894,E2 -28277.894} C_VEL
LIN {X 0,Y 124.78,Z 423.091,A -85,B 0,C 180,E1 -28279.55,E2 -28279.55} C_VEL
LIN {X 0,Y 117.364,Z 432.207,A -85,B 0,C 180,E1 -28281.849,E2 -28281.849} C_VEL
LIN {X 0,Y 108.449,Z 441.186,A -85,B 0,C 180,E1 -28284.869,E2 -28284.869} C_VEL
LIN {X 0,Y 99.955,Z 448.396,A -85,B 0,C 180,E1 -28288.491,E2 -28288.491} C_VEL
LIN {X 0,Y 92.002,Z 454.121,A -85,B 0,C 180,E1 -28292.829,E2 -28292.829} C_VEL
LIN {X 0,Y 84.607,Z 458.609,A -85,B 0,C 180,E1 -28297.895,E2 -28297.895} C_VEL
LIN {X 0,Y 77.969,Z 462.003,A -85,B 0,C 180,E1 -28303.854,E2 -28303.854} C_VEL
LIN {X 0,Y 70.638,Z 464.946,A -85,B 0,C 180,E1 -28313.348,E2 -28313.348} C_VEL
LIN {X 0,Y 67.694,Z 465.82,A -85,B 0,C 180,E1 -28318.728,E2 -28318.728} C_VEL
LIN {X 0,Y 65.357,Z 466.263,A -85,B 0,C 180,E1 -28324.524,E2 -28324.524} C_VEL
LIN {X 0,Y 62.752,Z 465.95,A -85,B 0,C 180,E1 -28337.056,E2 -28337.056} C_VEL
LIN {X 0,Y 62.438,Z 465.22,A -85,B 0,C 180,E1 -28343.537,E2 -28343.537} C_VEL
LIN {X 0,Y 62.687,Z 464.065,A -85,B 0,C 180,E1 -28350,E2 -28350} C_VEL
LIN {X 0,Y 64.126,Z 461.58,A -85,B 0,C 180,E1 -28359.465,E2 -28359.465} C_VEL
LIN {X 0,Y 66.843,Z 458.11,A -85,B 0,C 180,E1 -28368.386,E2 -28368.386} C_VEL
LIN {X 0,Y 70.908,Z 453.55,A -85,B 0,C 180,E1 -28376.488,E2 -28376.488} C_VEL
LIN {X 0,Y 77.089,Z 446.65,A -85,B 0,C 180,E1 -28384.736,E2 -28384.736} C_VEL
LIN {X 0,Y 83.329,Z 439.319,A -85,B 0,C 180,E1 -28390.657,E2 -28390.657} C_VEL
LIN {X 0,Y 89.258,Z 431.567,A -85,B 0,C 180,E1 -28395.124,E2 -28395.124} C_VEL
LIN {X 0,Y 95.539,Z 422.305,A -85,B 0,C 180,E1 -28398.938,E2 -28398.938} C_VEL
LIN {X 0,Y 101.481,Z 411.999,A -85,B 0,C 180,E1 -28401.977,E2 -28401.977} C_VEL
LIN {X 0,Y 106.93,Z 400.572,A -85,B 0,C 180,E1 -28404.424,E2 -28404.424} C_VEL
LIN {X 0,Y 111.05,Z 389.798,A -85,B 0,C 180,E1 -28406.106,E2 -28406.106} C_VEL
LIN {X 0,Y 114.67,Z 377.44,A -85,B 0,C 180,E1 -28407.46,E2 -28407.46} C_VEL
LIN {X 0,Y 117.276,Z 364.238,A -85,B 0,C 180,E1 -28408.431,E2 -28408.431} C_VEL
LIN {X 0,Y 120.025,Z 338.527,A -85,B 0,C 180,E1 -28409.483,E2 -28409.483} C_VEL
LIN {X 0,Y 117.295,Z 332.088,A -85,B 0,C 180,E1 -28413.142,E2 -28413.142} C_VEL
LIN {X 0,Y 114.666,Z 326.513,A -85,B 0,C 180,E1 -28417.356,E2 -28417.356} C_VEL
LIN {X 0,Y 112.575,Z 322.419,A -85,B 0,C 180,E1 -28421.592,E2 -28421.592} C_VEL
LIN {X 0,Y 110.848,Z 318.985,A -85,B 0,C 180,E1 -28426.491,E2 -28426.491} C_VEL
LIN {X 0,Y 109.485,Z 315.568,A -85,B 0,C 180,E1 -28436.319,E2 -28436.319} C_VEL
LIN {X 0,Y 109.54,Z 315.915,A -85,B 0,C 180,E1 -28439.31,E2 -28439.31} C_VEL
LIN {X 0,Y 110.942,Z 318.967,A -85,B 0,C 180,E1 -28447.416,E2 -28447.416} C_VEL
LIN {X 0,Y 113.039,Z 323.303,A -85,B 0,C 180,E1 -28453.096,E2 -28453.096} C_VEL
LIN {X 0,Y 115.055,Z 327.349,A -85,B 0,C 180,E1 -28456.981,E2 -28456.981} C_VEL
LIN {X 0,Y 117.296,Z 332.028,A -85,B 0,C 180,E1 -28460.496,E2 -28460.496} C_VEL
LIN {X 0,Y 119.091,Z 336.35,A -85,B 0,C 180,E1 -28462.986,E2 -28462.986} C_VEL
LIN {X 0,Y 119.979,Z 339.616,A -85,B 0,C 180,E1 -28464.26,E2 -28464.26} C_VEL
LIN {X 0,Y 117.11,Z 366.863,A -85,B 0,C 180,E1 -28465.365,E2 -28465.365} C_VEL
LIN {X 0,Y 114.289,Z 380.692,A -85,B 0,C 180,E1 -28466.283,E2 -28466.283} C_VEL
LIN {X 0,Y 110.505,Z 393.184,A -85,B 0,C 180,E1 -28467.575,E2 -28467.575} C_VEL
LIN {X 0,Y 105.812,Z 404.923,A -85,B 0,C 180,E1 -28469.336,E2 -28469.336} C_VEL
LIN {X 0,Y 100.181,Z 416.249,A -85,B 0,C 180,E1 -28471.723,E2 -28471.723} C_VEL
LIN {X 0,Y 94.071,Z 426.434,A -85,B 0,C 180,E1 -28474.735,E2 -28474.735} C_VEL
LIN {X 0,Y 87.667,Z 435.61,A -85,B 0,C 180,E1 -28478.591,E2 -28478.591} C_VEL
LIN {X 0,Y 80.497,Z 444.852,A -85,B 0,C 180,E1 -28484.303,E2 -28484.303} C_VEL
LIN {X 0,Y 75.649,Z 450.638,A -85,B 0,C 180,E1 -28489.435,E2 -28489.435} C_VEL
LIN {X 0,Y 70.321,Z 456.593,A -85,B 0,C 180,E1 -28496.655,E2 -28496.655} C_VEL
LIN {X 0,Y 66.227,Z 461.287,A -85,B 0,C 180,E1 -28504.883,E2 -28504.883} C_VEL
LIN {X 0,Y 63.713,Z 464.866,A -85,B 0,C 180,E1 -28513.993,E2 -28513.993} C_VEL
LIN {X 0,Y 62.587,Z 467.418,A -85,B 0,C 180,E1 -28523.553,E2 -28523.553} C_VEL
LIN {X 0,Y 62.612,Z 468.609,A -85,B 0,C 180,E1 -28530,E2 -28530} C_VEL
LIN {X 0,Y 62.645,Z 469.333,A -85,B 0,C 180,E1 -28536.442,E2 -28536.442} C_VEL
LIN {X 0,Y 64.494,Z 469.612,A -85,B 0,C 180,E1 -28549.082,E2 -28549.082} C_VEL
LIN {X 0,Y 66.451,Z 469.182,A -85,B 0,C 180,E1 -28555.027,E2 -28555.027} C_VEL
LIN {X 0,Y 69.027,Z 468.329,A -85,B 0,C 180,E1 -28560.603,E2 -28560.603} C_VEL
LIN {X 0,Y 76.088,Z 465.423,A -85,B 0,C 180,E1 -28570.283,E2 -28570.283} C_VEL
LIN {X 0,Y 82.611,Z 462.12,A -85,B 0,C 180,E1 -28576.314,E2 -28576.314} C_VEL
LIN {X 0,Y 89.795,Z 457.763,A -85,B 0,C 180,E1 -28581.506,E2 -28581.506} C_VEL
LIN {X 0,Y 97.6,Z 452.234,A -85,B 0,C 180,E1 -28585.903,E2 -28585.903} C_VEL
LIN {X 0,Y 105.999,Z 445.35,A -85,B 0,C 180,E1 -28589.535,E2 -28589.535} C_VEL
LIN {X 0,Y 114.821,Z 436.749,A -85,B 0,C 180,E1 -28592.563,E2 -28592.563} C_VEL
LIN {X 0,Y 122.324,Z 427.947,A -85,B 0,C 180,E1 -28594.81,E2 -28594.81} C_VEL
LIN {X 0,Y 130.093,Z 417.118,A -85,B 0,C 180,E1 -28596.692,E2 -28596.692} C_VEL
LIN {X 0,Y 136.406,Z 406.216,A -85,B 0,C 180,E1 -28598.035,E2 -28598.035} C_VEL
LIN {X 0,Y 141.95,Z 394.014,A -85,B 0,C 180,E1 -28599.149,E2 -28599.149} C_VEL
LIN {X 0,Y 146.143,Z 381.857,A -85,B 0,C 180,E1 -28599.931,E2 -28599.931} C_VEL
LIN {X 0,Y 149.174,Z 369.393,A -85,B 0,C 180,E1 -28600.434,E2 -28600.434} C_VEL
LIN {X 0,Y 149.793,Z 365.695,A -85,B 0,C 180,E1 -28600.594,E2 -28600.594} C_VEL
LIN {X 0,Y 148.623,Z 360.441,A -85,B 0,C 180,E1 -28603.429,E2 -28603.429} C_VEL
LIN {X 0,Y 147.114,Z 356.84,A -85,B 0,C 180,E1 -28607.06,E2 -28607.06} C_VEL
LIN {X 0,Y 146.295,Z 354.681,A -85,B 0,C 180,E1 -28609.797,E2 -28609.797} C_VEL
LIN {X 0,Y 145.497,Z 351.2,A -85,B 0,C 180,E1 -28616.539,E2 -28616.539} C_VEL
LIN {X 0,Y 145.531,Z 351.405,A -85,B 0,C 180,E1 -28618.963,E2 -28618.963} C_VEL
LIN {X 0,Y 145.617,Z 352.386,A -85,B 0,C 180,E1 -28620.71,E2 -28620.71} C_VEL
LIN {X 0,Y 145.718,Z 353.832,A -85,B 0,C 180,E1 -28622.153,E2 -28622.153} C_VEL
LIN {X 0,Y 145.799,Z 357.719,A -85,B 0,C 180,E1 -28624.272,E2 -28624.272} C_VEL
LIN {X 0,Y 145.949,Z 362.872,A -85,B 0,C 180,E1 -28626.749,E2 -28626.749} C_VEL
LIN {X 0,Y 146.086,Z 364.262,A -85,B 0,C 180,E1 -28627.657,E2 -28627.657} C_VEL
LIN {X 0,Y 147.262,Z 368.371,A -85,B 0,C 180,E1 -28631.284,E2 -28631.284} C_VEL
LIN {X 0,Y 144.092,Z 380.926,A -85,B 0,C 180,E1 -28631.914,E2 -28631.914} C_VEL
LIN {X 0,Y 139.945,Z 392.592,A -85,B 0,C 180,E1 -28632.717,E2 -28632.717} C_VEL
LIN {X 0,Y 134.737,Z 403.766,A -85,B 0,C 180,E1 -28633.713,E2 -28633.713} C_VEL
LIN {X 0,Y 128.259,Z 414.777,A -85,B 0,C 180,E1 -28635.035,E2 -28635.035} C_VEL
LIN {X 0,Y 121.25,Z 424.517,A -85,B 0,C 180,E1 -28636.726,E2 -28636.726} C_VEL
LIN {X 0,Y 113.34,Z 433.692,A -85,B 0,C 180,E1 -28638.982,E2 -28638.982} C_VEL
LIN {X 0,Y 104.121,Z 442.445,A -85,B 0,C 180,E1 -28641.859,E2 -28641.859} C_VEL
LIN {X 0,Y 95.289,Z 449.402,A -85,B 0,C 180,E1 -28645.378,E2 -28645.378} C_VEL
LIN {X 0,Y 85.606,Z 455.761,A -85,B 0,C 180,E1 -28650.456,E2 -28650.456} C_VEL
LIN {X 0,Y 77.869,Z 459.915,A -85,B 0,C 180,E1 -28655.68,E2 -28655.68} C_VEL
LIN {X 0,Y 73.157,Z 462.102,A -85,B 0,C 180,E1 -28659.777,E2 -28659.777} C_VEL
LIN {X 0,Y 65.775,Z 464.849,A -85,B 0,C 180,E1 -28668.413,E2 -28668.413} C_VEL
LIN {X 0,Y 61.659,Z 465.975,A -85,B 0,C 180,E1 -28675.256,E2 -28675.256} C_VEL
LIN {X 0,Y 58.973,Z 466.453,A -85,B 0,C 180,E1 -28681.53,E2 -28681.53} C_VEL
LIN {X 0,Y 55.788,Z 466.175,A -85,B 0,C 180,E1 -28695.407,E2 -28695.407} C_VEL
LIN {X 0,Y 55.346,Z 465.461,A -85,B 0,C 180,E1 -28702.704,E2 -28702.704} C_VEL
LIN {X 0,Y 55.58,Z 464.34,A -85,B 0,C 180,E1 -28710,E2 -28710} C_VEL
LIN {X 0,Y 56.462,Z 462.787,A -85,B 0,C 180,E1 -28717.15,E2 -28717.15} C_VEL
LIN {X 0,Y 59,Z 459.688,A -85,B 0,C 180,E1 -28727.325,E2 -28727.325} C_VEL
LIN {X 0,Y 63.002,Z 455.544,A -85,B 0,C 180,E1 -28736.5,E2 -28736.5} C_VEL
LIN {X 0,Y 69.321,Z 449.228,A -85,B 0,C 180,E1 -28745.659,E2 -28745.659} C_VEL
LIN {X 0,Y 75.85,Z 442.351,A -85,B 0,C 180,E1 -28752.203,E2 -28752.203} C_VEL
LIN {X 0,Y 83.153,Z 433.731,A -85,B 0,C 180,E1 -28757.692,E2 -28757.692} C_VEL
LIN {X 0,Y 89.716,Z 424.9,A -85,B 0,C 180,E1 -28761.569,E2 -28761.569} C_VEL
LIN {X 0,Y 95.885,Z 415.204,A -85,B 0,C 180,E1 -28764.629,E2 -28764.629} C_VEL
LIN {X 0,Y 101.536,Z 404.577,A -85,B 0,C 180,E1 -28767.061,E2 -28767.061} C_VEL
LIN {X 0,Y 106.604,Z 392.674,A -85,B 0,C 180,E1 -28768.986,E2 -28768.986} C_VEL
LIN {X 0,Y 110.658,Z 380.205,A -85,B 0,C 180,E1 -28770.407,E2 -28770.407} C_VEL
LIN {X 0,Y 113.488,Z 367.891,A -85,B 0,C 180,E1 -28771.371,E2 -28771.371} C_VEL
LIN {X 0,Y 115.391,Z 353.823,A -85,B 0,C 180,E1 -28772.015,E2 -28772.015} C_VEL
LIN {X 0,Y 116.614,Z 341.751,A -85,B 0,C 180,E1 -28772.459,E2 -28772.459} C_VEL
LIN {X 0,Y 113.935,Z 335.164,A -85,B 0,C 180,E1 -28776.797,E2 -28776.797} C_VEL
LIN {X 0,Y 112.12,Z 331.17,A -85,B 0,C 180,E1 -28780.395,E2 -28780.395} C_VEL
LIN {X 0,Y 111.001,Z 328.811,A -85,B 0,C 180,E1 -28783.109,E2 -28783.109} C_VEL
LIN {X 0,Y 109.654,Z 325.778,A -85,B 0,C 180,E1 -28787.532,E2 -28787.532} C_VEL
LIN {X 0,Y 108.605,Z 322.727,A -85,B 0,C 180,E1 -28796.289,E2 -28796.289} C_VEL
LIN {X 0,Y 108.653,Z 323.124,A -85,B 0,C 180,E1 -28799.305,E2 -28799.305} C_VEL
LIN {X 0,Y 109.765,Z 325.792,A -85,B 0,C 180,E1 -28806.468,E2 -28806.468} C_VEL
LIN {X 0,Y 111.585,Z 329.957,A -85,B 0,C 180,E1 -28811.999,E2 -28811.999} C_VEL
LIN {X 0,Y 113.598,Z 334.343,A -85,B 0,C 180,E1 -28816.222,E2 -28816.222} C_VEL
LIN {X 0,Y 115.977,Z 340.039,A -85,B 0,C 180,E1 -28820.218,E2 -28820.218} C_VEL
LIN {X 0,Y 116.628,Z 342.281,A -85,B 0,C 180,E1 -28821.279,E2 -28821.279} C_VEL
LIN {X 0,Y 113.882,Z 366.872,A -85,B 0,C 180,E1 -28822.227,E2 -28822.227} C_VEL
LIN {X 0,Y 110.972,Z 380.603,A -85,B 0,C 180,E1 -28823.088,E2 -28823.088} C_VEL
LIN {X 0,Y 107.016,Z 393.171,A -85,B 0,C 180,E1 -28824.328,E2 -28824.328} C_VEL
LIN {X 0,Y 101.755,Z 405.665,A -85,B 0,C 180,E1 -28826.119,E2 -28826.119} C_VEL
LIN {X 0,Y 95.889,Z 416.81,A -85,B 0,C 180,E1 -28828.416,E2 -28828.416} C_VEL
LIN {X 0,Y 90.198,Z 425.83,A -85,B 0,C 180,E1 -28831.009,E2 -28831.009} C_VEL
LIN {X 0,Y 83.393,Z 435.079,A -85,B 0,C 180,E1 -28834.747,E2 -28834.747} C_VEL
LIN {X 0,Y 75.809,Z 444.226,A -85,B 0,C 180,E1 -28840.316,E2 -28840.316} C_VEL
LIN {X 0,Y 70.401,Z 450.214,A -85,B 0,C 180,E1 -28845.67,E2 -28845.67} C_VEL
LIN {X 0,Y 64.478,Z 456.211,A -85,B 0,C 180,E1 -28853.167,E2 -28853.167} C_VEL
LIN {X 0,Y 59.829,Z 460.944,A -85,B 0,C 180,E1 -28861.974,E2 -28861.974} C_VEL
LIN {X 0,Y 56.899,Z 464.56,A -85,B 0,C 180,E1 -28872.014,E2 -28872.014} C_VEL
LIN {X 0,Y 55.537,Z 467.148,A -85,B 0,C 180,E1 -28882.73,E2 -28882.73} C_VEL
LIN {X 0,Y 55.511,Z 468.361,A -85,B 0,C 180,E1 -28890,E2 -28890} C_VEL
LIN {X 0,Y 55.583,Z 469.111,A -85,B 0,C 180,E1 -28897.264,E2 -28897.264} C_VEL
LIN {X 0,Y 57.821,Z 469.423,A -85,B 0,C 180,E1 -28911.386,E2 -28911.386} C_VEL
LIN {X 0,Y 60.054,Z 469.009,A -85,B 0,C 180,E1 -28917.912,E2 -28917.912} C_VEL
LIN {X 0,Y 63.001,Z 468.189,A -85,B 0,C 180,E1 -28923.902,E2 -28923.902} C_VEL
LIN {X 0,Y 70.795,Z 465.317,A -85,B 0,C 180,E1 -28934.02,E2 -28934.02} C_VEL
LIN {X 0,Y 77.858,Z 462.051,A -85,B 0,C 180,E1 -28940.109,E2 -28940.109} C_VEL
LIN {X 0,Y 85.545,Z 457.733,A -85,B 0,C 180,E1 -28945.241,E2 -28945.241} C_VEL
LIN {X 0,Y 95.231,Z 451.233,A -85,B 0,C 180,E1 -28950.129,E2 -28950.129} C_VEL
LIN {X 0,Y 104.091,Z 444.112,A -85,B 0,C 180,E1 -28953.459,E2 -28953.459} C_VEL
LIN {X 0,Y 113.258,Z 435.265,A -85,B 0,C 180,E1 -28956.246,E2 -28956.246} C_VEL
LIN {X 0,Y 121.063,Z 426.205,A -85,B 0,C 180,E1 -28958.255,E2 -28958.255} C_VEL
LIN {X 0,Y 128.274,Z 416.203,A -85,B 0,C 180,E1 -28959.762,E2 -28959.762} C_VEL
LIN {X 0,Y 134.738,Z 405.094,A -85,B 0,C 180,E1 -28960.981,E2 -28960.981} C_VEL
LIN {X 0,Y 140.392,Z 392.66,A -85,B 0,C 180,E1 -28962.015,E2 -28962.015} C_VEL
LIN {X 0,Y 144.705,Z 379.909,A -85,B 0,C 180,E1 -28962.72,E2 -28962.72} C_VEL
LIN {X 0,Y 147.276,Z 369.173,A -85,B 0,C 180,E1 -28963.125,E2 -28963.125} C_VEL
LIN {X 0,Y 146.755,Z 366.33,A -85,B 0,C 180,E1 -28964.907,E2 -28964.907} C_VEL
LIN {X 0,Y 145.829,Z 363.521,A -85,B 0,C 180,E1 -28967.828,E2 -28967.828} C_VEL
LIN {X 0,Y 145.144,Z 361.406,A -85,B 0,C 180,E1 -28970.595,E2 -28970.595} C_VEL
LIN {X 0,Y 144.627,Z 358.26,A -85,B 0,C 180,E1 -28976.518,E2 -28976.518} C_VEL
LIN {X 0,Y 144.632,Z 358.428,A -85,B 0,C 180,E1 -28978.608,E2 -28978.608} C_VEL
LIN {X 0,Y 145.339,Z 361.737,A -85,B 0,C 180,E1 -28984.681,E2 -28984.681} C_VEL
LIN {X 0,Y 146.086,Z 364.262,A -85,B 0,C 180,E1 -28987.657,E2 -28987.657} C_VEL
LIN {X 0,Y 146.119,Z 366.393,A -85,B 0,C 180,E1 -28988.56,E2 -28988.56} C_VEL
LIN {X 0,Y 145.775,Z 369.305,A -85,B 0,C 180,E1 -28989.099,E2 -28989.099} C_VEL
LIN {X 0,Y 144.958,Z 373.149,A -85,B 0,C 180,E1 -28989.362,E2 -28989.362} C_VEL
LIN {X 0,Y 141.332,Z 384.579,A -85,B 0,C 180,E1 -28989.365,E2 -28989.365} C_VEL
LIN {X 0,Y 136.301,Z 397.048,A -85,B 0,C 180,E1 -28990.176,E2 -28990.176} C_VEL
LIN {X 0,Y 129.918,Z 409.206,A -85,B 0,C 180,E1 -28991.338,E2 -28991.338} C_VEL
LIN {X 0,Y 123.3,Z 419.181,A -85,B 0,C 180,E1 -28992.549,E2 -28992.549} C_VEL
LIN {X 0,Y 115.987,Z 428.336,A -85,B 0,C 180,E1 -28994.19,E2 -28994.19} C_VEL
LIN {X 0,Y 108.012,Z 436.7,A -85,B 0,C 180,E1 -28996.314,E2 -28996.314} C_VEL
LIN {X 0,Y 98.551,Z 444.859,A -85,B 0,C 180,E1 -28999.108,E2 -28999.108} C_VEL
LIN {X 0,Y 90.927,Z 450.395,A -85,B 0,C 180,E1 -29001.949,E2 -29001.949} C_VEL
LIN {X 0,Y 82.184,Z 455.786,A -85,B 0,C 180,E1 -29006.114,E2 -29006.114} C_VEL
LIN {X 0,Y 73.9,Z 459.98,A -85,B 0,C 180,E1 -29011.138,E2 -29011.138} C_VEL
LIN {X 0,Y 68.777,Z 462.195,A -85,B 0,C 180,E1 -29015.166,E2 -29015.166} C_VEL
LIN {X 0,Y 60.001,Z 465.142,A -85,B 0,C 180,E1 -29024.652,E2 -29024.652} C_VEL
LIN {X 0,Y 55.902,Z 466.131,A -85,B 0,C 180,E1 -29031.053,E2 -29031.053} C_VEL
LIN {X 0,Y 52.765,Z 466.64,A -85,B 0,C 180,E1 -29037.806,E2 -29037.806} C_VEL
LIN {X 0,Y 48.895,Z 466.399,A -85,B 0,C 180,E1 -29053.293,E2 -29053.293} C_VEL
LIN {X 0,Y 48.283,Z 465.701,A -85,B 0,C 180,E1 -29061.63,E2 -29061.63} C_VEL
LIN {X 0,Y 48.464,Z 464.611,A -85,B 0,C 180,E1 -29070,E2 -29070} C_VEL
LIN {X 0,Y 49.442,Z 463.078,A -85,B 0,C 180,E1 -29078.172,E2 -29078.172} C_VEL
LIN {X 0,Y 51.623,Z 460.662,A -85,B 0,C 180,E1 -29087.634,E2 -29087.634} C_VEL
LIN {X 0,Y 56.757,Z 455.911,A -85,B 0,C 180,E1 -29099.69,E2 -29099.69} C_VEL
LIN {X 0,Y 63.7,Z 449.638,A -85,B 0,C 180,E1 -29109.375,E2 -29109.375} C_VEL
LIN {X 0,Y 70.769,Z 442.809,A -85,B 0,C 180,E1 -29116.054,E2 -29116.054} C_VEL
LIN {X 0,Y 78.578,Z 434.27,A -85,B 0,C 180,E1 -29121.498,E2 -29121.498} C_VEL
LIN {X 0,Y 85.503,Z 425.509,A -85,B 0,C 180,E1 -29125.281,E2 -29125.281} C_VEL
LIN {X 0,Y 92.701,Z 414.729,A -85,B 0,C 180,E1 -29128.528,E2 -29128.528} C_VEL
LIN {X 0,Y 98.626,Z 403.883,A -85,B 0,C 180,E1 -29130.8,E2 -29130.8} C_VEL
LIN {X 0,Y 103.835,Z 391.908,A -85,B 0,C 180,E1 -29132.574,E2 -29132.574} C_VEL
LIN {X 0,Y 108,Z 379.292,A -85,B 0,C 180,E1 -29133.883,E2 -29133.883} C_VEL
LIN {X 0,Y 110.885,Z 366.547,A -85,B 0,C 180,E1 -29134.757,E2 -29134.757} C_VEL
LIN {X 0,Y 113.002,Z 350.25,A -85,B 0,C 180,E1 -29135.391,E2 -29135.391} C_VEL
LIN {X 0,Y 113.468,Z 345.033,A -85,B 0,C 180,E1 -29135.681,E2 -29135.681} C_VEL
LIN {X 0,Y 111.297,Z 339.371,A -85,B 0,C 180,E1 -29139.998,E2 -29139.998} C_VEL
LIN {X 0,Y 109.72,Z 335.549,A -85,B 0,C 180,E1 -29144.061,E2 -29144.061} C_VEL
LIN {X 0,Y 108.558,Z 332.63,A -85,B 0,C 180,E1 -29148.353,E2 -29148.353} C_VEL
LIN {X 0,Y 107.731,Z 329.847,A -85,B 0,C 180,E1 -29156.259,E2 -29156.259} C_VEL
LIN {X 0,Y 107.751,Z 330.053,A -85,B 0,C 180,E1 -29158.598,E2 -29158.598} C_VEL
LIN {X 0,Y 108.666,Z 332.703,A -85,B 0,C 180,E1 -29165.701,E2 -29165.701} C_VEL
LIN {X 0,Y 110.128,Z 336.462,A -85,B 0,C 180,E1 -29170.74,E2 -29170.74} C_VEL
LIN {X 0,Y 112.018,Z 341.074,A -85,B 0,C 180,E1 -29175.173,E2 -29175.173} C_VEL
LIN {X 0,Y 113.574,Z 345.314,A -85,B 0,C 180,E1 -29178.151,E2 -29178.151} C_VEL
LIN {X 0,Y 111.004,Z 366.977,A -85,B 0,C 180,E1 -29178.932,E2 -29178.932} C_VEL
LIN {X 0,Y 108.012,Z 380.567,A -85,B 0,C 180,E1 -29179.725,E2 -29179.725} C_VEL
LIN {X 0,Y 103.891,Z 393.146,A -85,B 0,C 180,E1 -29180.871,E2 -29180.871} C_VEL
LIN {X 0,Y 98.827,Z 404.811,A -85,B 0,C 180,E1 -29182.41,E2 -29182.41} C_VEL
LIN {X 0,Y 92.693,Z 416.082,A -85,B 0,C 180,E1 -29184.517,E2 -29184.517} C_VEL
LIN {X 0,Y 86.004,Z 426.217,A -85,B 0,C 180,E1 -29187.294,E2 -29187.294} C_VEL
LIN {X 0,Y 78.156,Z 436.184,A -85,B 0,C 180,E1 -29191.322,E2 -29191.322} C_VEL
LIN {X 0,Y 70.244,Z 444.963,A -85,B 0,C 180,E1 -29196.831,E2 -29196.831} C_VEL
LIN {X 0,Y 64.301,Z 450.91,A -85,B 0,C 180,E1 -29202.459,E2 -29202.459} C_VEL
LIN {X 0,Y 58.921,Z 455.827,A -85,B 0,C 180,E1 -29209.002,E2 -29209.002} C_VEL
LIN {X 0,Y 53.628,Z 460.599,A -85,B 0,C 180,E1 -29218.385,E2 -29218.385} C_VEL
LIN {X 0,Y 50.151,Z 464.253,A -85,B 0,C 180,E1 -29229.492,E2 -29229.492} C_VEL
LIN {X 0,Y 48.491,Z 466.877,A -85,B 0,C 180,E1 -29241.667,E2 -29241.667} C_VEL
LIN {X 0,Y 48.428,Z 468.108,A -85,B 0,C 180,E1 -29250,E2 -29250} C_VEL
LIN {X 0,Y 48.551,Z 468.89,A -85,B 0,C 180,E1 -29258.323,E2 -29258.323} C_VEL
LIN {X 0,Y 51.238,Z 469.234,A -85,B 0,C 180,E1 -29274.299,E2 -29274.299} C_VEL
LIN {X 0,Y 57.231,Z 468.048,A -85,B 0,C 180,E1 -29287.88,E2 -29287.88} C_VEL
LIN {X 0,Y 65.854,Z 465.212,A -85,B 0,C 180,E1 -29298.335,E2 -29298.335} C_VEL
LIN {X 0,Y 73.493,Z 461.983,A -85,B 0,C 180,E1 -29304.375,E2 -29304.375} C_VEL
LIN {X 0,Y 81.685,Z 457.703,A -85,B 0,C 180,E1 -29309.359,E2 -29309.359} C_VEL
LIN {X 0,Y 91.902,Z 451.249,A -85,B 0,C 180,E1 -29313.969,E2 -29313.969} C_VEL
LIN {X 0,Y 101.117,Z 444.196,A -85,B 0,C 180,E1 -29317.061,E2 -29317.061} C_VEL
LIN {X 0,Y 110.588,Z 435.405,A -85,B 0,C 180,E1 -29319.616,E2 -29319.616} C_VEL
LIN {X 0,Y 119.44,Z 425.433,A -85,B 0,C 180,E1 -29321.59,E2 -29321.59} C_VEL
LIN {X 0,Y 126.814,Z 415.254,A -85,B 0,C 180,E1 -29322.938,E2 -29322.938} C_VEL
LIN {X 0,Y 133.422,Z 403.976,A -85,B 0,C 180,E1 -29324.012,E2 -29324.012} C_VEL
LIN {X 0,Y 138.914,Z 391.98,A -85,B 0,C 180,E1 -29324.891,E2 -29324.891} C_VEL
LIN {X 0,Y 143.289,Z 379.047,A -85,B 0,C 180,E1 -29325.512,E2 -29325.512} C_VEL
LIN {X 0,Y 144.863,Z 372.79,A -85,B 0,C 180,E1 -29325.783,E2 -29325.783} C_VEL
LIN {X 0,Y 144.084,Z 369.568,A -85,B 0,C 180,E1 -29329.327,E2 -29329.327} C_VEL
LIN {X 0,Y 143.769,Z 368.186,A -85,B 0,C 180,E1 -29331.213,E2 -29331.213} C_VEL
LIN {X 0,Y 143.517,Z 365.208,A -85,B 0,C 180,E1 -29337.193,E2 -29337.193} C_VEL
LIN {X 0,Y 143.479,Z 365.59,A -85,B 0,C 180,E1 -29338.597,E2 -29338.597} C_VEL
LIN {X 0,Y 143.894,Z 368.632,A -85,B 0,C 180,E1 -29344.202,E2 -29344.202} C_VEL
LIN {X 0,Y 144.481,Z 371.851,A -85,B 0,C 180,E1 -29347.776,E2 -29347.776} C_VEL
LIN {X 0,Y 144.709,Z 372.815,A -85,B 0,C 180,E1 -29348.73,E2 -29348.73} C_VEL
LIN {X 0,Y 141.332,Z 384.579,A -85,B 0,C 180,E1 -29349.365,E2 -29349.365} C_VEL
LIN {X 0,Y 139.841,Z 388.279,A -85,B 0,C 180,E1 -29349.274,E2 -29349.274} C_VEL
LIN {X 0,Y 133.772,Z 399.762,A -85,B 0,C 180,E1 -29347.696,E2 -29347.696} C_VEL
LIN {X 0,Y 131.849,Z 403.232,A -85,B 0,C 180,E1 -29347.7,E2 -29347.7} C_VEL
LIN {X 0,Y 125.323,Z 414.111,A -85,B 0,C 180,E1 -29348.737,E2 -29348.737} C_VEL
LIN {X 0,Y 118.6,Z 423.235,A -85,B 0,C 180,E1 -29349.889,E2 -29349.889} C_VEL
LIN {X 0,Y 111.149,Z 431.734,A -85,B 0,C 180,E1 -29351.456,E2 -29351.456} C_VEL
LIN {X 0,Y 102.932,Z 439.546,A -85,B 0,C 180,E1 -29353.354,E2 -29353.354} C_VEL
LIN {X 0,Y 93.238,Z 447.154,A -85,B 0,C 180,E1 -29356.041,E2 -29356.041} C_VEL
LIN {X 0,Y 82.93,Z 453.794,A -85,B 0,C 180,E1 -29359.816,E2 -29359.816} C_VEL
LIN {X 0,Y 73.355,Z 458.781,A -85,B 0,C 180,E1 -29364.471,E2 -29364.471} C_VEL
LIN {X 0,Y 64.887,Z 462.282,A -85,B 0,C 180,E1 -29369.946,E2 -29369.946} C_VEL
LIN {X 0,Y 59.659,Z 464.041,A -85,B 0,C 180,E1 -29374.45,E2 -29374.45} C_VEL
LIN {X 0,Y 50.518,Z 466.287,A -85,B 0,C 180,E1 -29385.926,E2 -29385.926} C_VEL
LIN {X 0,Y 46.845,Z 466.821,A -85,B 0,C 180,E1 -29393.122,E2 -29393.122} C_VEL
LIN {X 0,Y 42.066,Z 466.623,A -85,B 0,C 180,E1 -29410.48,E2 -29410.48} C_VEL
LIN {X 0,Y 41.229,Z 465.942,A -85,B 0,C 180,E1 -29420.185,E2 -29420.185} C_VEL
LIN {X 0,Y 41.339,Z 464.877,A -85,B 0,C 180,E1 -29430,E2 -29430} C_VEL
LIN {X 0,Y 42.43,Z 463.369,A -85,B 0,C 180,E1 -29439.534,E2 -29439.534} C_VEL
LIN {X 0,Y 46.461,Z 459.663,A -85,B 0,C 180,E1 -29454.822,E2 -29454.822} C_VEL
LIN {X 0,Y 52.746,Z 454.672,A -85,B 0,C 180,E1 -29466.84,E2 -29466.84} C_VEL
LIN {X 0,Y 59.609,Z 449.044,A -85,B 0,C 180,E1 -29475.024,E2 -29475.024} C_VEL
LIN {X 0,Y 67.405,Z 441.986,A -85,B 0,C 180,E1 -29481.443,E2 -29481.443} C_VEL
LIN {X 0,Y 75.803,Z 433.192,A -85,B 0,C 180,E1 -29486.555,E2 -29486.555} C_VEL
LIN {X 0,Y 83.923,Z 423.186,A -85,B 0,C 180,E1 -29490.323,E2 -29490.323} C_VEL
LIN {X 0,Y 90.746,Z 412.949,A -85,B 0,C 180,E1 -29492.953,E2 -29492.953} C_VEL
LIN {X 0,Y 96.937,Z 401.6,A -85,B 0,C 180,E1 -29494.993,E2 -29494.993} C_VEL
LIN {X 0,Y 102.168,Z 389.378,A -85,B 0,C 180,E1 -29496.556,E2 -29496.556} C_VEL
LIN {X 0,Y 106.18,Z 376.669,A -85,B 0,C 180,E1 -29497.626,E2 -29497.626} C_VEL
LIN {X 0,Y 108.903,Z 363.846,A -85,B 0,C 180,E1 -29498.369,E2 -29498.369} C_VEL
LIN {X 0,Y 110.743,Z 348.814,A -85,B 0,C 180,E1 -29498.901,E2 -29498.901} C_VEL
LIN {X 0,Y 109.095,Z 344.023,A -85,B 0,C 180,E1 -29503.066,E2 -29503.066} C_VEL
LIN {X 0,Y 108.238,Z 341.773,A -85,B 0,C 180,E1 -29505.813,E2 -29505.813} C_VEL
LIN {X 0,Y 107.458,Z 339.438,A -85,B 0,C 180,E1 -29509.32,E2 -29509.32} C_VEL
LIN {X 0,Y 106.852,Z 336.993,A -85,B 0,C 180,E1 -29516.228,E2 -29516.228} C_VEL
LIN {X 0,Y 106.866,Z 337.111,A -85,B 0,C 180,E1 -29518.292,E2 -29518.292} C_VEL
LIN {X 0,Y 107.526,Z 339.459,A -85,B 0,C 180,E1 -29524.61,E2 -29524.61} C_VEL
LIN {X 0,Y 108.747,Z 343.06,A -85,B 0,C 180,E1 -29529.527,E2 -29529.527} C_VEL
LIN {X 0,Y 110.252,Z 347.267,A -85,B 0,C 180,E1 -29533.595,E2 -29533.595} C_VEL
LIN {X 0,Y 110.788,Z 348.878,A -85,B 0,C 180,E1 -29534.828,E2 -29534.828} C_VEL
LIN {X 0,Y 108.367,Z 367.878,A -85,B 0,C 180,E1 -29535.502,E2 -29535.502} C_VEL
LIN {X 0,Y 105.477,Z 380.391,A -85,B 0,C 180,E1 -29536.169,E2 -29536.169} C_VEL
LIN {X 0,Y 101.572,Z 392.123,A -85,B 0,C 180,E1 -29537.116,E2 -29537.116} C_VEL
LIN {X 0,Y 96.34,Z 403.957,A -85,B 0,C 180,E1 -29538.495,E2 -29538.495} C_VEL
LIN {X 0,Y 89.971,Z 415.348,A -85,B 0,C 180,E1 -29540.386,E2 -29540.386} C_VEL
LIN {X 0,Y 82.965,Z 425.609,A -85,B 0,C 180,E1 -29542.895,E2 -29542.895} C_VEL
LIN {X 0,Y 74.688,Z 435.647,A -85,B 0,C 180,E1 -29546.629,E2 -29546.629} C_VEL
LIN {X 0,Y 66.202,Z 444.493,A -85,B 0,C 180,E1 -29551.866,E2 -29551.866} C_VEL
LIN {X 0,Y 59.734,Z 450.482,A -85,B 0,C 180,E1 -29557.423,E2 -29557.423} C_VEL
LIN {X 0,Y 53.736,Z 455.441,A -85,B 0,C 180,E1 -29564.001,E2 -29564.001} C_VEL
LIN {X 0,Y 47.691,Z 460.253,A -85,B 0,C 180,E1 -29573.881,E2 -29573.881} C_VEL
LIN {X 0,Y 43.533,Z 463.945,A -85,B 0,C 180,E1 -29586.197,E2 -29586.197} C_VEL
LIN {X 0,Y 41.46,Z 466.605,A -85,B 0,C 180,E1 -29600.241,E2 -29600.241} C_VEL
LIN {X 0,Y 41.327,Z 467.853,A -85,B 0,C 180,E1 -29610,E2 -29610} C_VEL
LIN {X 0,Y 41.53,Z 468.667,A -85,B 0,C 180,E1 -29619.743,E2 -29619.743} C_VEL
LIN {X 0,Y 44.828,Z 469.045,A -85,B 0,C 180,E1 -29638.056,E2 -29638.056} C_VEL
LIN {X 0,Y 51.801,Z 467.902,A -85,B 0,C 180,E1 -29652.716,E2 -29652.716} C_VEL
LIN {X 0,Y 56.365,Z 466.708,A -85,B 0,C 180,E1 -29658.429,E2 -29658.429} C_VEL
LIN {X 0,Y 64.032,Z 464.173,A -85,B 0,C 180,E1 -29665.405,E2 -29665.405} C_VEL
LIN {X 0,Y 73.586,Z 460.075,A -85,B 0,C 180,E1 -29671.476,E2 -29671.476} C_VEL
LIN {X 0,Y 84.357,Z 454.22,A -85,B 0,C 180,E1 -29676.411,E2 -29676.411} C_VEL
LIN {X 0,Y 93.744,Z 447.963,A -85,B 0,C 180,E1 -29679.575,E2 -29679.575} C_VEL
LIN {X 0,Y 103.433,Z 440.147,A -85,B 0,C 180,E1 -29682.039,E2 -29682.039} C_VEL
LIN {X 0,Y 111.612,Z 432.191,A -85,B 0,C 180,E1 -29683.794,E2 -29683.794} C_VEL
LIN {X 0,Y 119.073,Z 423.561,A -85,B 0,C 180,E1 -29685.127,E2 -29685.127} C_VEL
LIN {X 0,Y 126.596,Z 413.015,A -85,B 0,C 180,E1 -29686.292,E2 -29686.292} C_VEL
LIN {X 0,Y 133.341,Z 401.236,A -85,B 0,C 180,E1 -29687.183,E2 -29687.183} C_VEL
LIN {X 0,Y 138.517,Z 389.381,A -85,B 0,C 180,E1 -29687.901,E2 -29687.901} C_VEL
LIN {X 0,Y 142.415,Z 377.456,A -85,B 0,C 180,E1 -29688.394,E2 -29688.394} C_VEL
LIN {X 0,Y 142.069,Z 374.976,A -85,B 0,C 180,E1 -29691.643,E2 -29691.643} C_VEL
LIN {X 0,Y 142.014,Z 372.219,A -85,B 0,C 180,E1 -29697.164,E2 -29697.164} C_VEL
LIN {X 0,Y 141.902,Z 372.951,A -85,B 0,C 180,E1 -29699.113,E2 -29699.113} C_VEL
LIN {X 0,Y 142.037,Z 375.317,A -85,B 0,C 180,E1 -29703.546,E2 -29703.546} C_VEL
LIN {X 0,Y 142.25,Z 377.43,A -85,B 0,C 180,E1 -29706.118,E2 -29706.118} C_VEL
LIN {X 0,Y 138.356,Z 389.167,A -85,B 0,C 180,E1 -29706.764,E2 -29706.764} C_VEL
LIN {X 0,Y 132.925,Z 401.211,A -85,B 0,C 180,E1 -29707.543,E2 -29707.543} C_VEL
LIN {X 0,Y 131.849,Z 403.232,A -85,B 0,C 180,E1 -29707.7,E2 -29707.7} C_VEL
LIN {X 0,Y 128.885,Z 408.334,A -85,B 0,C 180,E1 -29707.861,E2 -29707.861} C_VEL
LIN {X 0,Y 123.217,Z 416.406,A -85,B 0,C 180,E1 -29707.371,E2 -29707.371} C_VEL
LIN {X 0,Y 116.928,Z 423.992,A -85,B 0,C 180,E1 -29706.914,E2 -29706.914} C_VEL
LIN {X 0,Y 112.976,Z 428.327,A -85,B 0,C 180,E1 -29707.204,E2 -29707.204} C_VEL
LIN {X 0,Y 104.897,Z 436.46,A -85,B 0,C 180,E1 -29708.796,E2 -29708.796} C_VEL
LIN {X 0,Y 94.823,Z 444.727,A -85,B 0,C 180,E1 -29710.87,E2 -29710.87} C_VEL
LIN {X 0,Y 86.582,Z 450.359,A -85,B 0,C 180,E1 -29713.078,E2 -29713.078} C_VEL
LIN {X 0,Y 76.858,Z 455.878,A -85,B 0,C 180,E1 -29716.466,E2 -29716.466} C_VEL
LIN {X 0,Y 67.591,Z 460.111,A -85,B 0,C 180,E1 -29720.641,E2 -29720.641} C_VEL
LIN {X 0,Y 61.606,Z 462.367,A -85,B 0,C 180,E1 -29724.128,E2 -29724.128} C_VEL
LIN {X 0,Y 55.898,Z 464.162,A -85,B 0,C 180,E1 -29728.344,E2 -29728.344} C_VEL
LIN {X 0,Y 45.635,Z 466.443,A -85,B 0,C 180,E1 -29739.643,E2 -29739.643} C_VEL
LIN {X 0,Y 41.331,Z 466.996,A -85,B 0,C 180,E1 -29747.143,E2 -29747.143} C_VEL
LIN {X 0,Y 37.803,Z 467.129,A -85,B 0,C 180,E1 -29756.1,E2 -29756.1} C_VEL
LIN {X 0,Y 34.198,Z 466.183,A -85,B 0,C 180,E1 -29778.14,E2 -29778.14} C_VEL
LIN {X 0,Y 34.216,Z 465.136,A -85,B 0,C 180,E1 -29790,E2 -29790} C_VEL
LIN {X 0,Y 35.444,Z 463.661,A -85,B 0,C 180,E1 -29801.436,E2 -29801.436} C_VEL
LIN {X 0,Y 39.215,Z 460.672,A -85,B 0,C 180,E1 -29816.618,E2 -29816.618} C_VEL
LIN {X 0,Y 45.002,Z 456.645,A -85,B 0,C 180,E1 -29828.659,E2 -29828.659} C_VEL
LIN {X 0,Y 53.528,Z 450.456,A -85,B 0,C 180,E1 -29839.02,E2 -29839.02} C_VEL
LIN {X 0,Y 61.807,Z 443.721,A -85,B 0,C 180,E1 -29845.527,E2 -29845.527} C_VEL
LIN {X 0,Y 70.652,Z 435.35,A -85,B 0,C 180,E1 -29850.504,E2 -29850.504} C_VEL
LIN {X 0,Y 78.313,Z 426.727,A -85,B 0,C 180,E1 -29853.82,E2 -29853.82} C_VEL
LIN {X 0,Y 86.177,Z 416.113,A -85,B 0,C 180,E1 -29856.559,E2 -29856.559} C_VEL
LIN {X 0,Y 92.559,Z 405.566,A -85,B 0,C 180,E1 -29858.457,E2 -29858.457} C_VEL
LIN {X 0,Y 98.123,Z 394.034,A -85,B 0,C 180,E1 -29859.888,E2 -29859.888} C_VEL
LIN {X 0,Y 102.417,Z 382.407,A -85,B 0,C 180,E1 -29860.927,E2 -29860.927} C_VEL
LIN {X 0,Y 105.729,Z 369.857,A -85,B 0,C 180,E1 -29861.743,E2 -29861.743} C_VEL
LIN {X 0,Y 107.906,Z 356.6,A -85,B 0,C 180,E1 -29862.213,E2 -29862.213} C_VEL
LIN {X 0,Y 108.313,Z 352.591,A -85,B 0,C 180,E1 -29862.423,E2 -29862.423} C_VEL
LIN {X 0,Y 107.128,Z 348.746,A -85,B 0,C 180,E1 -29866.484,E2 -29866.484} C_VEL
LIN {X 0,Y 106.327,Z 346.143,A -85,B 0,C 180,E1 -29870.672,E2 -29870.672} C_VEL
LIN {X 0,Y 105.972,Z 344.158,A -85,B 0,C 180,E1 -29876.197,E2 -29876.197} C_VEL
LIN {X 0,Y 105.988,Z 344.069,A -85,B 0,C 180,E1 -29877.684,E2 -29877.684} C_VEL
LIN {X 0,Y 106.49,Z 346.475,A -85,B 0,C 180,E1 -29883.929,E2 -29883.929} C_VEL
LIN {X 0,Y 107.455,Z 349.785,A -85,B 0,C 180,E1 -29888.426,E2 -29888.426} C_VEL
LIN {X 0,Y 108.354,Z 352.716,A -85,B 0,C 180,E1 -29891.338,E2 -29891.338} C_VEL
LIN {X 0,Y 106.174,Z 368.564,A -85,B 0,C 180,E1 -29891.903,E2 -29891.903} C_VEL
LIN {X 0,Y 103.303,Z 380.446,A -85,B 0,C 180,E1 -29892.467,E2 -29892.467} C_VEL
LIN {X 0,Y 99.293,Z 392.099,A -85,B 0,C 180,E1 -29893.289,E2 -29893.289} C_VEL
LIN {X 0,Y 93.492,Z 404.691,A -85,B 0,C 180,E1 -29894.571,E2 -29894.571} C_VEL
LIN {X 0,Y 86.929,Z 415.913,A -85,B 0,C 180,E1 -29896.246,E2 -29896.246} C_VEL
LIN {X 0,Y 79.656,Z 425.99,A -85,B 0,C 180,E1 -29898.475,E2 -29898.475} C_VEL
LIN {X 0,Y 71.774,Z 435.111,A -85,B 0,C 180,E1 -29901.53,E2 -29901.53} C_VEL
LIN {X 0,Y 62.721,Z 444.014,A -85,B 0,C 180,E1 -29906.311,E2 -29906.311} C_VEL
LIN {X 0,Y 54.296,Z 451.144,A -85,B 0,C 180,E1 -29912.718,E2 -29912.718} C_VEL
LIN {X 0,Y 46.6,Z 456.817,A -85,B 0,C 180,E1 -29921.056,E2 -29921.056} C_VEL
LIN {X 0,Y 40.235,Z 461.279,A -85,B 0,C 180,E1 -29932.313,E2 -29932.313} C_VEL
LIN {X 0,Y 35.959,Z 464.658,A -85,B 0,C 180,E1 -29946.991,E2 -29946.991} C_VEL
LIN {X 0,Y 34.478,Z 466.333,A -85,B 0,C 180,E1 -29958.239,E2 -29958.239} C_VEL
LIN {X 0,Y 34.241,Z 467.599,A -85,B 0,C 180,E1 -29970,E2 -29970} C_VEL
LIN {X 0,Y 34.537,Z 468.438,A -85,B 0,C 180,E1 -29981.742,E2 -29981.742} C_VEL
LIN {X 0,Y 38.682,Z 468.856,A -85,B 0,C 180,E1 -30003.03,E2 -30003.03} C_VEL
LIN {X 0,Y 46.827,Z 467.75,A -85,B 0,C 180,E1 -30018.627,E2 -30018.627} C_VEL
LIN {X 0,Y 51.919,Z 466.586,A -85,B 0,C 180,E1 -30024.311,E2 -30024.311} C_VEL
LIN {X 0,Y 57.385,Z 465.003,A -85,B 0,C 180,E1 -30029.016,E2 -30029.016} C_VEL
LIN {X 0,Y 67.596,Z 461.266,A -85,B 0,C 180,E1 -30035.21,E2 -30035.21} C_VEL
LIN {X 0,Y 78.581,Z 456.017,A -85,B 0,C 180,E1 -30039.899,E2 -30039.899} C_VEL
LIN {X 0,Y 89.865,Z 449.114,A -85,B 0,C 180,E1 -30043.341,E2 -30043.341} C_VEL
LIN {X 0,Y 99.803,Z 441.655,A -85,B 0,C 180,E1 -30045.525,E2 -30045.525} C_VEL
LIN {X 0,Y 108.147,Z 434.061,A -85,B 0,C 180,E1 -30047.107,E2 -30047.107} C_VEL
LIN {X 0,Y 116.605,Z 424.865,A -85,B 0,C 180,E1 -30048.357,E2 -30048.357} C_VEL
LIN {X 0,Y 124.253,Z 414.642,A -85,B 0,C 180,E1 -30049.347,E2 -30049.347} C_VEL
LIN {X 0,Y 131.099,Z 403.31,A -85,B 0,C 180,E1 -30050.083,E2 -30050.083} C_VEL
LIN {X 0,Y 136.586,Z 391.676,A -85,B 0,C 180,E1 -30050.728,E2 -30050.728} C_VEL
LIN {X 0,Y 139.387,Z 384.215,A -85,B 0,C 180,E1 -30050.967,E2 -30050.967} C_VEL
LIN {X 0,Y 139.956,Z 382.241,A -85,B 0,C 180,E1 -30051.336,E2 -30051.336} C_VEL
LIN {X 0,Y 140.08,Z 379.317,A -85,B 0,C 180,E1 -30057.124,E2 -30057.124} C_VEL
LIN {X 0,Y 139.876,Z 380.396,A -85,B 0,C 180,E1 -30060,E2 -30060} C_VEL
LIN {X 0,Y 139.84,Z 382.197,A -85,B 0,C 180,E1 -30063.266,E2 -30063.266} C_VEL
LIN {X 0,Y 139.311,Z 383.998,A -85,B 0,C 180,E1 -30063.592,E2 -30063.592} C_VEL
LIN {X 0,Y 134.522,Z 395.917,A -85,B 0,C 180,E1 -30064.18,E2 -30064.18} C_VEL
LIN {X 0,Y 128.731,Z 406.94,A -85,B 0,C 180,E1 -30064.898,E2 -30064.898} C_VEL
LIN {X 0,Y 121.857,Z 417.404,A -85,B 0,C 180,E1 -30065.798,E2 -30065.798} C_VEL
LIN {X 0,Y 113.328,Z 427.952,A -85,B 0,C 180,E1 -30067.145,E2 -30067.145} C_VEL
LIN {X 0,Y 112.976,Z 428.327,A -85,B 0,C 180,E1 -30067.204,E2 -30067.204} C_VEL
LIN {X 0,Y 108.821,Z 432.569,A -85,B 0,C 180,E1 -30067.558,E2 -30067.558} C_VEL
LIN {X 0,Y 98.218,Z 441.494,A -85,B 0,C 180,E1 -30067.106,E2 -30067.106} C_VEL
LIN {X 0,Y 91.807,Z 446.09,A -85,B 0,C 180,E1 -30067.151,E2 -30067.151} C_VEL
LIN {X 0,Y 88.606,Z 448.208,A -85,B 0,C 180,E1 -30067.615,E2 -30067.615} C_VEL
LIN {X 0,Y 77.584,Z 454.688,A -85,B 0,C 180,E1 -30070.439,E2 -30070.439} C_VEL
LIN {X 0,Y 68.652,Z 458.873,A -85,B 0,C 180,E1 -30073.461,E2 -30073.461} C_VEL
LIN {X 0,Y 59.034,Z 462.451,A -85,B 0,C 180,E1 -30077.747,E2 -30077.747} C_VEL
LIN {X 0,Y 52.857,Z 464.281,A -85,B 0,C 180,E1 -30081.449,E2 -30081.449} C_VEL
LIN {X 0,Y 41.425,Z 466.598,A -85,B 0,C 180,E1 -30091.974,E2 -30091.974} C_VEL
LIN {X 0,Y 36.405,Z 467.168,A -85,B 0,C 180,E1 -30099.448,E2 -30099.448} C_VEL
LIN {X 0,Y 32.095,Z 467.336,A -85,B 0,C 180,E1 -30108.934,E2 -30108.934} C_VEL
LIN {X 0,Y 27.246,Z 466.423,A -85,B 0,C 180,E1 -30135.051,E2 -30135.051} C_VEL
LIN {X 0,Y 27.078,Z 465.394,A -85,B 0,C 180,E1 -30149.999,E2 -30149.999} C_VEL
LIN {X 0,Y 28.503,Z 463.953,A -85,B 0,C 180,E1 -30164.274,E2 -30164.274} C_VEL
LIN {X 0,Y 33.031,Z 460.996,A -85,B 0,C 180,E1 -30182.135,E2 -30182.135} C_VEL
LIN {X 0,Y 39.731,Z 457.005,A -85,B 0,C 180,E1 -30195.037,E2 -30195.037} C_VEL
LIN {X 0,Y 49.18,Z 450.865,A -85,B 0,C 180,E1 -30205.255,E2 -30205.255} C_VEL
LIN {X 0,Y 58.098,Z 444.178,A -85,B 0,C 180,E1 -30211.285,E2 -30211.285} C_VEL
LIN {X 0,Y 67.453,Z 435.88,A -85,B 0,C 180,E1 -30215.736,E2 -30215.736} C_VEL
LIN {X 0,Y 75.466,Z 427.335,A -85,B 0,C 180,E1 -30218.634,E2 -30218.634} C_VEL
LIN {X 0,Y 83.615,Z 416.807,A -85,B 0,C 180,E1 -30221.011,E2 -30221.011} C_VEL
LIN {X 0,Y 90.206,Z 406.365,A -85,B 0,C 180,E1 -30222.631,E2 -30222.631} C_VEL
LIN {X 0,Y 95.912,Z 395.104,A -85,B 0,C 180,E1 -30223.835,E2 -30223.835} C_VEL
LIN {X 0,Y 100.211,Z 384.099,A -85,B 0,C 180,E1 -30224.701,E2 -30224.701} C_VEL
LIN {X 0,Y 103.976,Z 370.562,A -85,B 0,C 180,E1 -30225.485,E2 -30225.485} C_VEL
LIN {X 0,Y 106.227,Z 357.594,A -85,B 0,C 180,E1 -30225.885,E2 -30225.885} C_VEL
LIN {X 0,Y 106.255,Z 356.717,A -85,B 0,C 180,E1 -30226.125,E2 -30226.125} C_VEL
LIN {X 0,Y 105.491,Z 353.733,A -85,B 0,C 180,E1 -30230.17,E2 -30230.17} C_VEL
LIN {X 0,Y 105.088,Z 351.35,A -85,B 0,C 180,E1 -30236.165,E2 -30236.165} C_VEL
LIN {X 0,Y 105.129,Z 351.884,A -85,B 0,C 180,E1 -30239.521,E2 -30239.521} C_VEL
LIN {X 0,Y 105.428,Z 353.235,A -85,B 0,C 180,E1 -30242.865,E2 -30242.865} C_VEL
LIN {X 0,Y 106.184,Z 356.43,A -85,B 0,C 180,E1 -30247.212,E2 -30247.212} C_VEL
LIN {X 0,Y 106.322,Z 356.966,A -85,B 0,C 180,E1 -30247.799,E2 -30247.799} C_VEL
LIN {X 0,Y 104.041,Z 370.963,A -85,B 0,C 180,E1 -30248.241,E2 -30248.241} C_VEL
LIN {X 0,Y 100.614,Z 383.444,A -85,B 0,C 180,E1 -30248.743,E2 -30248.743} C_VEL
LIN {X 0,Y 96.206,Z 395.076,A -85,B 0,C 180,E1 -30249.531,E2 -30249.531} C_VEL
LIN {X 0,Y 90.273,Z 406.973,A -85,B 0,C 180,E1 -30250.615,E2 -30250.615} C_VEL
LIN {X 0,Y 82.697,Z 418.805,A -85,B 0,C 180,E1 -30252.226,E2 -30252.226} C_VEL
LIN {X 0,Y 74.387,Z 429.304,A -85,B 0,C 180,E1 -30254.44,E2 -30254.44} C_VEL
LIN {X 0,Y 66.241,Z 437.797,A -85,B 0,C 180,E1 -30257.278,E2 -30257.278} C_VEL
LIN {X 0,Y 57.208,Z 445.758,A -85,B 0,C 180,E1 -30261.626,E2 -30261.626} C_VEL
LIN {X 0,Y 49.304,Z 451.752,A -85,B 0,C 180,E1 -30267.015,E2 -30267.015} C_VEL
LIN {X 0,Y 39.627,Z 458.08,A -85,B 0,C 180,E1 -30277.052,E2 -30277.052} C_VEL
LIN {X 0,Y 32.818,Z 462.208,A -85,B 0,C 180,E1 -30290.026,E2 -30290.026} C_VEL
LIN {X 0,Y 29.518,Z 464.368,A -85,B 0,C 180,E1 -30301.564,E2 -30301.564} C_VEL
LIN {X 0,Y 27.545,Z 466.06,A -85,B 0,C 180,E1 -30315.218,E2 -30315.218} C_VEL
LIN {X 0,Y 27.127,Z 467.344,A -85,B 0,C 180,E1 -30330.001,E2 -30330.001} C_VEL
LIN {X 0,Y 27.62,Z 468.204,A -85,B 0,C 180,E1 -30344.742,E2 -30344.742} C_VEL
LIN {X 0,Y 29.602,Z 468.636,A -85,B 0,C 180,E1 -30358.349,E2 -30358.349} C_VEL
LIN {X 0,Y 37.301,Z 468.319,A -85,B 0,C 180,E1 -30378.909,E2 -30378.909} C_VEL
LIN {X 0,Y 42.468,Z 467.595,A -85,B 0,C 180,E1 -30385.838,E2 -30385.838} C_VEL
LIN {X 0,Y 48.111,Z 466.464,A -85,B 0,C 180,E1 -30391.22,E2 -30391.22} C_VEL
LIN {X 0,Y 54.068,Z 464.899,A -85,B 0,C 180,E1 -30395.492,E2 -30395.492} C_VEL
LIN {X 0,Y 66.058,Z 460.758,A -85,B 0,C 180,E1 -30401.388,E2 -30401.388} C_VEL
LIN {X 0,Y 76.429,Z 455.995,A -85,B 0,C 180,E1 -30404.913,E2 -30404.913} C_VEL
LIN {X 0,Y 88.091,Z 449.149,A -85,B 0,C 180,E1 -30407.775,E2 -30407.775} C_VEL
LIN {X 0,Y 98.271,Z 441.739,A -85,B 0,C 180,E1 -30409.53,E2 -30409.53} C_VEL
LIN {X 0,Y 108.512,Z 432.535,A -85,B 0,C 180,E1 -30411.004,E2 -30411.004} C_VEL
LIN {X 0,Y 116.25,Z 424.051,A -85,B 0,C 180,E1 -30411.878,E2 -30411.878} C_VEL
LIN {X 0,Y 124.009,Z 413.689,A -85,B 0,C 180,E1 -30412.652,E2 -30412.652} C_VEL
LIN {X 0,Y 130.74,Z 402.541,A -85,B 0,C 180,E1 -30413.209,E2 -30413.209} C_VEL
LIN {X 0,Y 136.195,Z 390.986,A -85,B 0,C 180,E1 -30413.726,E2 -30413.726} C_VEL
LIN {X 0,Y 136.865,Z 389.278,A -85,B 0,C 180,E1 -30413.76,E2 -30413.76} C_VEL
LIN {X 0,Y 137.449,Z 387.63,A -85,B 0,C 180,E1 -30414.131,E2 -30414.131} C_VEL
LIN {X 0,Y 137.743,Z 386.214,A -85,B 0,C 180,E1 -30417.076,E2 -30417.076} C_VEL
LIN {X 0,Y 137.41,Z 387.583,A -85,B 0,C 180,E1 -30420.733,E2 -30420.733} C_VEL
LIN {X 0,Y 132.581,Z 398.629,A -85,B 0,C 180,E1 -30421.276,E2 -30421.276} C_VEL
LIN {X 0,Y 126.574,Z 409.398,A -85,B 0,C 180,E1 -30421.9,E2 -30421.9} C_VEL
LIN {X 0,Y 118.733,Z 420.557,A -85,B 0,C 180,E1 -30422.734,E2 -30422.734} C_VEL
LIN {X 0,Y 109.606,Z 430.949,A -85,B 0,C 180,E1 -30423.963,E2 -30423.963} C_VEL
LIN {X 0,Y 100.595,Z 439.323,A -85,B 0,C 180,E1 -30425.394,E2 -30425.394} C_VEL
LIN {X 0,Y 90.326,Z 447.072,A -85,B 0,C 180,E1 -30427.235,E2 -30427.235} C_VEL
LIN {X 0,Y 88.606,Z 448.208,A -85,B 0,C 180,E1 -30427.615,E2 -30427.615} C_VEL
LIN {X 0,Y 83.637,Z 451.27,A -85,B 0,C 180,E1 -30428.285,E2 -30428.285} C_VEL
LIN {X 0,Y 74.823,Z 455.857,A -85,B 0,C 180,E1 -30428.352,E2 -30428.352} C_VEL
LIN {X 0,Y 65.689,Z 459.693,A -85,B 0,C 180,E1 -30428.544,E2 -30428.544} C_VEL
LIN {X 0,Y 60.248,Z 461.578,A -85,B 0,C 180,E1 -30429.725,E2 -30429.725} C_VEL
LIN {X 0,Y 50.673,Z 464.393,A -85,B 0,C 180,E1 -30433.867,E2 -30433.867} C_VEL
LIN {X 0,Y 41.411,Z 466.285,A -85,B 0,C 180,E1 -30439.843,E2 -30439.843} C_VEL
LIN {X 0,Y 32.314,Z 467.342,A -85,B 0,C 180,E1 -30449.546,E2 -30449.546} C_VEL
LIN {X 0,Y 27.103,Z 467.538,A -85,B 0,C 180,E1 -30458.929,E2 -30458.929} C_VEL
LIN {X 0,Y 22.956,Z 467.296,A -85,B 0,C 180,E1 -30472.244,E2 -30472.244} C_VEL
LIN {X 0,Y 20.407,Z 466.664,A -85,B 0,C 180,E1 -30489.855,E2 -30489.855} C_VEL
LIN {X 0,Y 19.96,Z 465.651,A -85,B 0,C 180,E1 -30509.999,E2 -30509.999} C_VEL
LIN {X 0,Y 21.694,Z 464.241,A -85,B 0,C 180,E1 -30528.902,E2 -30528.902} C_VEL
LIN {X 0,Y 27.298,Z 461.313,A -85,B 0,C 180,E1 -30550.063,E2 -30550.063} C_VEL
LIN {X 0,Y 35.09,Z 457.359,A -85,B 0,C 180,E1 -30563.238,E2 -30563.238} C_VEL
LIN {X 0,Y 45.514,Z 451.275,A -85,B 0,C 180,E1 -30572.607,E2 -30572.607} C_VEL
LIN {X 0,Y 55.048,Z 444.634,A -85,B 0,C 180,E1 -30577.76,E2 -30577.76} C_VEL
LIN {X 0,Y 64.869,Z 436.397,A -85,B 0,C 180,E1 -30581.438,E2 -30581.438} C_VEL
LIN {X 0,Y 73.186,Z 427.942,A -85,B 0,C 180,E1 -30583.798,E2 -30583.798} C_VEL
LIN {X 0,Y 81.59,Z 417.5,A -85,B 0,C 180,E1 -30585.709,E2 -30585.709} C_VEL
LIN {X 0,Y 89.209,Z 405.739,A -85,B 0,C 180,E1 -30587.141,E2 -30587.141} C_VEL
LIN {X 0,Y 94.87,Z 394.57,A -85,B 0,C 180,E1 -30588.069,E2 -30588.069} C_VEL
LIN {X 0,Y 99.56,Z 382.429,A -85,B 0,C 180,E1 -30588.806,E2 -30588.806} C_VEL
LIN {X 0,Y 103.122,Z 369.398,A -85,B 0,C 180,E1 -30589.383,E2 -30589.383} C_VEL
LIN {X 0,Y 104.551,Z 361.528,A -85,B 0,C 180,E1 -30589.653,E2 -30589.653} C_VEL
LIN {X 0,Y 104.269,Z 359.73,A -85,B 0,C 180,E1 -30592.739,E2 -30592.739} C_VEL
LIN {X 0,Y 104.191,Z 358.559,A -85,B 0,C 180,E1 -30596.132,E2 -30596.132} C_VEL
LIN {X 0,Y 104.217,Z 358.863,A -85,B 0,C 180,E1 -30599.034,E2 -30599.034} C_VEL
LIN {X 0,Y 104.388,Z 360.27,A -85,B 0,C 180,E1 -30602.17,E2 -30602.17} C_VEL
LIN {X 0,Y 104.592,Z 361.518,A -85,B 0,C 180,E1 -30604.093,E2 -30604.093} C_VEL
LIN {X 0,Y 102.108,Z 374.134,A -85,B 0,C 180,E1 -30604.458,E2 -30604.458} C_VEL
LIN {X 0,Y 98.338,Z 386.41,A -85,B 0,C 180,E1 -30604.859,E2 -30604.859} C_VEL
LIN {X 0,Y 93.558,Z 397.852,A -85,B 0,C 180,E1 -30605.539,E2 -30605.539} C_VEL
